LIN {X 0,Y 357.391,Z 435.676,A -85,B 0,C 180,E1 11294.259,E2 11294.259} C_VEL
LIN {X 0,Y 359.556,Z 438.789,A -85,B 0,C 180,E1 11291.438,E2 11291.438} C_VEL
LIN {X 0,Y 362.294,Z 441.241,A -85,B 0,C 180,E1 11287.88,E2 11287.88} C_VEL
LIN {X 0,Y 364.705,Z 442.533,A -85,B 0,C 180,E1 11284.575,E2 11284.575} C_VEL
LIN {X 0,Y 365.647,Z 443.721,A -85,B 0,C 180,E1 11283.201,E2 11283.201} C_VEL
LIN {X 0,Y 367.504,Z 446.415,A -85,B 0,C 180,E1 11280.039,E2 11280.039} C_VEL
LIN {X 0,Y 369.353,Z 448.083,A -85,B 0,C 180,E1 11276.876,E2 11276.876} C_VEL
LIN {X 0,Y 371.438,Z 449.318,A -85,B 0,C 180,E1 11272.974,E2 11272.974} C_VEL
LIN {X 0,Y 372.957,Z 450.083,A -85,B 0,C 180,E1 11269.742,E2 11269.742} C_VEL
LIN {X 0,Y 374.216,Z 452.056,A -85,B 0,C 180,E1 11266.292,E2 11266.292} C_VEL
LIN {X 0,Y 375.116,Z 453.423,A -85,B 0,C 180,E1 11263.095,E2 11263.095} C_VEL
LIN {X 0,Y 375.998,Z 454.396,A -85,B 0,C 180,E1 11259.644,E2 11259.644} C_VEL
LIN {X 0,Y 376.539,Z 454.956,A -85,B 0,C 180,E1 11256.097,E2 11256.097} C_VEL
LIN {X 0,Y 376.912,Z 455.194,A -85,B 0,C 180,E1 11252.737,E2 11252.737} C_VEL
LIN {X 0,Y 376.943,Z 455.24,A -85,B 0,C 180,E1 11249.088,E2 11249.088} C_VEL
LIN {X 0,Y 376.782,Z 455.124,A -85,B 0,C 180,E1 11245.739,E2 11245.739} C_VEL
LIN {X 0,Y 376.258,Z 454.711,A -85,B 0,C 180,E1 11242.057,E2 11242.057} C_VEL
LIN {X 0,Y 375.613,Z 454.001,A -85,B 0,C 180,E1 11238.795,E2 11238.795} C_VEL
LIN {X 0,Y 374.6,Z 452.721,A -85,B 0,C 180,E1 11235.066,E2 11235.066} C_VEL
LIN {X 0,Y 373.634,Z 450.999,A -85,B 0,C 180,E1 11232.077,E2 11232.077} C_VEL
LIN {X 0,Y 372.596,Z 449.782,A -85,B 0,C 180,E1 11229.419,E2 11229.419} C_VEL
LIN {X 0,Y 370.725,Z 448.948,A -85,B 0,C 180,E1 11225.63,E2 11225.63} C_VEL
LIN {X 0,Y 368.919,Z 447.787,A -85,B 0,C 180,E1 11222.391,E2 11222.391} C_VEL
LIN {X 0,Y 366.884,Z 445.572,A -85,B 0,C 180,E1 11218.816,E2 11218.816} C_VEL
LIN {X 0,Y 364.823,Z 442.577,A -85,B 0,C 180,E1 11215.582,E2 11215.582} C_VEL
LIN {X 0,Y 362.364,Z 441.294,A -85,B 0,C 180,E1 11212.227,E2 11212.227} C_VEL
LIN {X 0,Y 359.63,Z 438.864,A -85,B 0,C 180,E1 11208.648,E2 11208.648} C_VEL
LIN {X 0,Y 357.486,Z 435.84,A -85,B 0,C 180,E1 11205.86,E2 11205.86} C_VEL
LIN {X 0,Y 355.327,Z 434.438,A -85,B 0,C 180,E1 11203.361,E2 11203.361} C_VEL
LIN {X 0,Y 352.433,Z 432.047,A -85,B 0,C 180,E1 11200.091,E2 11200.091} C_VEL
LIN {X 0,Y 350.007,Z 428.702,A -85,B 0,C 180,E1 11197.273,E2 11197.273} C_VEL
LIN {X 0,Y 348.432,Z 427.598,A -85,B 0,C 180,E1 11195.628,E2 11195.628} C_VEL
LIN {X 0,Y 345.313,Z 425.117,A -85,B 0,C 180,E1 11192.389,E2 11192.389} C_VEL
LIN {X 0,Y 342.845,Z 421.896,A -85,B 0,C 180,E1 11189.721,E2 11189.721} C_VEL
LIN {X 0,Y 341.776,Z 420.845,A -85,B 0,C 180,E1 11188.671,E2 11188.671} C_VEL
LIN {X 0,Y 338.023,Z 418.479,A -85,B 0,C 180,E1 11185.586,E2 11185.586} C_VEL
LIN {X 0,Y 334.266,Z 415.023,A -85,B 0,C 180,E1 11182.883,E2 11182.883} C_VEL
LIN {X 0,Y 332.281,Z 413.005,A -85,B 0,C 180,E1 11181.537,E2 11181.537} C_VEL
LIN {X 0,Y 327.822,Z 409.906,A -85,B 0,C 180,E1 11178.863,E2 11178.863} C_VEL
LIN {X 0,Y 322.978,Z 404.536,A -85,B 0,C 180,E1 11175.687,E2 11175.687} C_VEL
LIN {X 0,Y 319.536,Z 400.127,A -85,B 0,C 180,E1 11172.836,E2 11172.836} C_VEL
LIN {X 0,Y 318.657,Z 398.667,A -85,B 0,C 180,E1 11171.952,E2 11171.952} C_VEL
LIN {X 0,Y 315.762,Z 394.618,A -85,B 0,C 180,E1 11168.467,E2 11168.467} C_VEL
LIN {X 0,Y 315.284,Z 393.503,A -85,B 0,C 180,E1 11167.654,E2 11167.654} C_VEL
LIN {X 0,Y 312.928,Z 391.284,A -85,B 0,C 180,E1 11160.915,E2 11160.915} C_VEL
LIN {X 0,Y 313.352,Z 391.949,A -85,B 0,C 180,E1 11156.891,E2 11156.891} C_VEL
LIN {X 0,Y 315.434,Z 393.763,A -85,B 0,C 180,E1 11152.533,E2 11152.533} C_VEL
LIN {X 0,Y 317.844,Z 397.884,A -85,B 0,C 180,E1 11149.304,E2 11149.304} C_VEL
LIN {X 0,Y 319.163,Z 399.431,A -85,B 0,C 180,E1 11147.976,E2 11147.976} C_VEL
LIN {X 0,Y 323.04,Z 405.209,A -85,B 0,C 180,E1 11144.655,E2 11144.655} C_VEL
LIN {X 0,Y 326.338,Z 410.188,A -85,B 0,C 180,E1 11142.343,E2 11142.343} C_VEL
LIN {X 0,Y 331.124,Z 417.365,A -85,B 0,C 180,E1 11139.496,E2 11139.496} C_VEL
LIN {X 0,Y 334.176,Z 422.791,A -85,B 0,C 180,E1 11137.852,E2 11137.852} C_VEL
LIN {X 0,Y 338.881,Z 432.418,A -85,B 0,C 180,E1 11135.51,E2 11135.51} C_VEL
LIN {X 0,Y 340.966,Z 437.107,A -85,B 0,C 180,E1 11134.535,E2 11134.535} C_VEL
LIN {X 0,Y 339.393,Z 457.12,A -85,B 0,C 180,E1 11134.133,E2 11134.133} C_VEL
LIN {X 0,Y 338.344,Z 464.817,A -85,B 0,C 180,E1 11134.132,E2 11134.132} C_VEL
LIN {X 0,Y 333.991,Z 485.367,A -85,B 0,C 180,E1 11134.678,E2 11134.678} C_VEL
LIN {X 0,Y 333.138,Z 491.97,A -85,B 0,C 180,E1 11134.661,E2 11134.661} C_VEL
LIN {X 0,Y 324.438,Z 599.073,A -85,B 0,C 180,E1 11132.465,E2 11132.465} C_VEL
LIN {X 0,Y 320.784,Z 623.389,A -85,B 0,C 180,E1 11131.786,E2 11131.786} C_VEL
LIN {X 0,Y 316.917,Z 641.647,A -85,B 0,C 180,E1 11131.101,E2 11131.101} C_VEL
LIN {X 0,Y 312.027,Z 660.593,A -85,B 0,C 180,E1 11130.177,E2 11130.177} C_VEL
LIN {X 0,Y 305.137,Z 682.435,A -85,B 0,C 180,E1 11128.783,E2 11128.783} C_VEL
LIN {X 0,Y 298.819,Z 699.564,A -85,B 0,C 180,E1 11127.404,E2 11127.404} C_VEL
LIN {X 0,Y 291.032,Z 718.423,A -85,B 0,C 180,E1 11125.539,E2 11125.539} C_VEL
LIN {X 0,Y 282.813,Z 735.832,A -85,B 0,C 180,E1 11123.371,E2 11123.371} C_VEL
LIN {X 0,Y 275.348,Z 750.463,A -85,B 0,C 180,E1 11121.158,E2 11121.158} C_VEL
LIN {X 0,Y 266.704,Z 766.363,A -85,B 0,C 180,E1 11118.247,E2 11118.247} C_VEL
LIN {X 0,Y 257.927,Z 781.243,A -85,B 0,C 180,E1 11114.814,E2 11114.814} C_VEL
LIN {X 0,Y 251.129,Z 792.469,A -85,B 0,C 180,E1 11111.673,E2 11111.673} C_VEL
LIN {X 0,Y 243.527,Z 804.944,A -85,B 0,C 180,E1 11107.419,E2 11107.419} C_VEL
LIN {X 0,Y 237.187,Z 815.301,A -85,B 0,C 180,E1 11102.942,E2 11102.942} C_VEL
LIN {X 0,Y 232.588,Z 823.275,A -85,B 0,C 180,E1 11098.722,E2 11098.722} C_VEL
LIN {X 0,Y 228.301,Z 831.546,A -85,B 0,C 180,E1 11093.213,E2 11093.213} C_VEL
LIN {X 0,Y 225.883,Z 837.101,A -85,B 0,C 180,E1 11088.317,E2 11088.317} C_VEL
LIN {X 0,Y 224.59,Z 841.14,A -85,B 0,C 180,E1 11083.647,E2 11083.647} C_VEL
LIN {X 0,Y 224.047,Z 844.149,A -85,B 0,C 180,E1 11078.727,E2 11078.727} C_VEL
LIN {X 0,Y 223.976,Z 845.889,A -85,B 0,C 180,E1 11073.583,E2 11073.583} C_VEL
LIN {X 0,Y 223.996,Z 846.17,A -85,B 0,C 180,E1 11068.977,E2 11068.977} C_VEL
LIN {X 0,Y 223.975,Z 845.377,A -85,B 0,C 180,E1 11064.563,E2 11064.563} C_VEL
LIN {X 0,Y 224.105,Z 843.591,A -85,B 0,C 180,E1 11060.239,E2 11060.239} C_VEL
LIN {X 0,Y 224.692,Z 840.748,A -85,B 0,C 180,E1 11055.834,E2 11055.834} C_VEL
LIN {X 0,Y 226.189,Z 836.341,A -85,B 0,C 180,E1 11050.907,E2 11050.907} C_VEL
LIN {X 0,Y 229.32,Z 829.45,A -85,B 0,C 180,E1 11045.256,E2 11045.256} C_VEL
LIN {X 0,Y 233.115,Z 822.315,A -85,B 0,C 180,E1 11040.729,E2 11040.729} C_VEL
LIN {X 0,Y 238.319,Z 813.453,A -85,B 0,C 180,E1 11036.171,E2 11036.171} C_VEL
LIN {X 0,Y 245.397,Z 801.813,A -85,B 0,C 180,E1 11031.437,E2 11031.437} C_VEL
LIN {X 0,Y 252.004,Z 791.031,A -85,B 0,C 180,E1 11027.894,E2 11027.894} C_VEL
LIN {X 0,Y 259.516,Z 778.645,A -85,B 0,C 180,E1 11024.524,E2 11024.524} C_VEL
LIN {X 0,Y 268.58,Z 762.891,A -85,B 0,C 180,E1 11021.076,E2 11021.076} C_VEL
LIN {X 0,Y 276.219,Z 748.803,A -85,B 0,C 180,E1 11018.569,E2 11018.569} C_VEL
LIN {X 0,Y 284.677,Z 732.136,A -85,B 0,C 180,E1 11016.119,E2 11016.119} C_VEL
LIN {X 0,Y 292.974,Z 713.8,A -85,B 0,C 180,E1 11013.975,E2 11013.975} C_VEL
LIN {X 0,Y 299.637,Z 697.472,A -85,B 0,C 180,E1 11012.413,E2 11012.413} C_VEL
LIN {X 0,Y 306.898,Z 677.436,A -85,B 0,C 180,E1 11010.857,E2 11010.857} C_VEL
LIN {X 0,Y 312.927,Z 657.297,A -85,B 0,C 180,E1 11009.65,E2 11009.65} C_VEL
LIN {X 0,Y 317.385,Z 639.669,A -85,B 0,C 180,E1 11008.816,E2 11008.816} C_VEL
LIN {X 0,Y 321.862,Z 617.639,A -85,B 0,C 180,E1 11008.03,E2 11008.03} C_VEL
LIN {X 0,Y 324.697,Z 596.376,A -85,B 0,C 180,E1 11007.475,E2 11007.475} C_VEL
LIN {X 0,Y 337.198,Z 440.954,A -85,B 0,C 180,E1 11004.294,E2 11004.294} C_VEL
LIN {X 0,Y 332.27,Z 430.413,A -85,B 0,C 180,E1 11001.77,E2 11001.77} C_VEL
LIN {X 0,Y 329.221,Z 424.769,A -85,B 0,C 180,E1 11000.071,E2 11000.071} C_VEL
LIN {X 0,Y 324.819,Z 417.96,A -85,B 0,C 180,E1 10997.373,E2 10997.373} C_VEL
LIN {X 0,Y 322.038,Z 413.675,A -85,B 0,C 180,E1 10995.394,E2 10995.394} C_VEL
LIN {X 0,Y 320.191,Z 410.862,A -85,B 0,C 180,E1 10993.913,E2 10993.913} C_VEL
LIN {X 0,Y 317.215,Z 406.295,A -85,B 0,C 180,E1 10991.085,E2 10991.085} C_VEL
LIN {X 0,Y 314.43,Z 402.015,A -85,B 0,C 180,E1 10987.491,E2 10987.491} C_VEL
LIN {X 0,Y 313.894,Z 401.23,A -85,B 0,C 180,E1 10986.585,E2 10986.585} C_VEL
LIN {X 0,Y 311.948,Z 399.214,A -85,B 0,C 180,E1 10980.367,E2 10980.367} C_VEL
LIN {X 0,Y 312.409,Z 399.942,A -85,B 0,C 180,E1 10976.33,E2 10976.33} C_VEL
LIN {X 0,Y 314.345,Z 401.757,A -85,B 0,C 180,E1 10972.231,E2 10972.231} C_VEL
LIN {X 0,Y 316.81,Z 405.872,A -85,B 0,C 180,E1 10968.9,E2 10968.9} C_VEL
LIN {X 0,Y 317.925,Z 407.334,A -85,B 0,C 180,E1 10967.744,E2 10967.744} C_VEL
LIN {X 0,Y 321.341,Z 412.052,A -85,B 0,C 180,E1 10964.756,E2 10964.756} C_VEL
LIN {X 0,Y 323.001,Z 413.964,A -85,B 0,C 180,E1 10963.546,E2 10963.546} C_VEL
LIN {X 0,Y 327.432,Z 418.519,A -85,B 0,C 180,E1 10960.744,E2 10960.744} C_VEL
LIN {X 0,Y 332.012,Z 421.761,A -85,B 0,C 180,E1 10957.98,E2 10957.98} C_VEL
LIN {X 0,Y 335.685,Z 425.45,A -85,B 0,C 180,E1 10955.355,E2 10955.355} C_VEL
LIN {X 0,Y 339.012,Z 427.854,A -85,B 0,C 180,E1 10952.797,E2 10952.797} C_VEL
LIN {X 0,Y 341.404,Z 429.368,A -85,B 0,C 180,E1 10950.72,E2 10950.72} C_VEL
LIN {X 0,Y 343.92,Z 432.708,A -85,B 0,C 180,E1 10948.054,E2 10948.054} C_VEL
LIN {X 0,Y 347.005,Z 435.312,A -85,B 0,C 180,E1 10944.811,E2 10944.811} C_VEL
LIN {X 0,Y 348.8,Z 436.444,A -85,B 0,C 180,E1 10942.988,E2 10942.988} C_VEL
LIN {X 0,Y 351.378,Z 439.984,A -85,B 0,C 180,E1 10939.978,E2 10939.978} C_VEL
LIN {X 0,Y 354.275,Z 442.359,A -85,B 0,C 180,E1 10936.701,E2 10936.701} C_VEL
LIN {X 0,Y 356.338,Z 443.696,A -85,B 0,C 180,E1 10934.315,E2 10934.315} C_VEL
LIN {X 0,Y 358.427,Z 446.646,A -85,B 0,C 180,E1 10931.598,E2 10931.598} C_VEL
LIN {X 0,Y 361.149,Z 449.073,A -85,B 0,C 180,E1 10928.124,E2 10928.124} C_VEL
LIN {X 0,Y 363.636,Z 450.443,A -85,B 0,C 180,E1 10924.691,E2 10924.691} C_VEL
LIN {X 0,Y 364.634,Z 451.698,A -85,B 0,C 180,E1 10923.245,E2 10923.245} C_VEL
LIN {X 0,Y 366.572,Z 454.443,A -85,B 0,C 180,E1 10919.943,E2 10919.943} C_VEL
LIN {X 0,Y 368.437,Z 456.074,A -85,B 0,C 180,E1 10916.769,E2 10916.769} C_VEL
LIN {X 0,Y 370.437,Z 457.251,A -85,B 0,C 180,E1 10913.015,E2 10913.015} C_VEL
LIN {X 0,Y 371.948,Z 458.011,A -85,B 0,C 180,E1 10909.798,E2 10909.798} C_VEL
LIN {X 0,Y 373.203,Z 459.944,A -85,B 0,C 180,E1 10906.439,E2 10906.439} C_VEL
LIN {X 0,Y 374.126,Z 461.361,A -85,B 0,C 180,E1 10903.13,E2 10903.13} C_VEL
LIN {X 0,Y 374.962,Z 462.31,A -85,B 0,C 180,E1 10899.826,E2 10899.826} C_VEL
LIN {X 0,Y 375.545,Z 462.87,A -85,B 0,C 180,E1 10896.267,E2 10896.267} C_VEL
LIN {X 0,Y 375.886,Z 463.11,A -85,B 0,C 180,E1 10893.049,E2 10893.049} C_VEL
LIN {X 0,Y 375.975,Z 463.189,A -85,B 0,C 180,E1 10889.238,E2 10889.238} C_VEL
LIN {X 0,Y 375.805,Z 463.095,A -85,B 0,C 180,E1 10886.034,E2 10886.034} C_VEL
LIN {X 0,Y 375.311,Z 462.674,A -85,B 0,C 180,E1 10882.191,E2 10882.191} C_VEL
LIN {X 0,Y 374.684,Z 462.013,A -85,B 0,C 180,E1 10879.079,E2 10879.079} C_VEL
LIN {X 0,Y 373.799,Z 460.907,A -85,B 0,C 180,E1 10875.534,E2 10875.534} C_VEL
LIN {X 0,Y 372.703,Z 459.108,A -85,B 0,C 180,E1 10872.244,E2 10872.244} C_VEL
LIN {X 0,Y 371.727,Z 457.816,A -85,B 0,C 180,E1 10869.698,E2 10869.698} C_VEL
LIN {X 0,Y 370.035,Z 457.027,A -85,B 0,C 180,E1 10866.09,E2 10866.09} C_VEL
LIN {X 0,Y 368.084,Z 455.848,A -85,B 0,C 180,E1 10862.655,E2 10862.655} C_VEL
LIN {X 0,Y 366.169,Z 453.933,A -85,B 0,C 180,E1 10859.296,E2 10859.296} C_VEL
LIN {X 0,Y 363.981,Z 450.622,A -85,B 0,C 180,E1 10855.776,E2 10855.776} C_VEL
LIN {X 0,Y 361.582,Z 449.398,A -85,B 0,C 180,E1 10852.525,E2 10852.525} C_VEL
LIN {X 0,Y 358.842,Z 447.06,A -85,B 0,C 180,E1 10848.886,E2 10848.886} C_VEL
LIN {X 0,Y 356.443,Z 443.873,A -85,B 0,C 180,E1 10845.817,E2 10845.817} C_VEL
LIN {X 0,Y 355.498,Z 442.991,A -85,B 0,C 180,E1 10844.638,E2 10844.638} C_VEL
LIN {X 0,Y 352.409,Z 440.929,A -85,B 0,C 180,E1 10841.165,E2 10841.165} C_VEL
LIN {X 0,Y 349.883,Z 438.191,A -85,B 0,C 180,E1 10838.325,E2 10838.325} C_VEL
LIN {X 0,Y 348.298,Z 435.966,A -85,B 0,C 180,E1 10836.458,E2 10836.458} C_VEL
LIN {X 0,Y 345.092,Z 433.842,A -85,B 0,C 180,E1 10833.203,E2 10833.203} C_VEL
LIN {X 0,Y 342.244,Z 430.64,A -85,B 0,C 180,E1 10830.148,E2 10830.148} C_VEL
LIN {X 0,Y 340.87,Z 428.854,A -85,B 0,C 180,E1 10828.754,E2 10828.754} C_VEL
LIN {X 0,Y 336.984,Z 426.486,A -85,B 0,C 180,E1 10825.582,E2 10825.582} C_VEL
LIN {X 0,Y 333.203,Z 423.143,A -85,B 0,C 180,E1 10822.876,E2 10822.876} C_VEL
LIN {X 0,Y 330.785,Z 420.741,A -85,B 0,C 180,E1 10821.267,E2 10821.267} C_VEL
LIN {X 0,Y 326.293,Z 417.595,A -85,B 0,C 180,E1 10818.583,E2 10818.583} C_VEL
LIN {X 0,Y 321.458,Z 412.16,A -85,B 0,C 180,E1 10815.33,E2 10815.33} C_VEL
LIN {X 0,Y 318.01,Z 407.503,A -85,B 0,C 180,E1 10812.345,E2 10812.345} C_VEL
LIN {X 0,Y 317.151,Z 406.22,A -85,B 0,C 180,E1 10811.456,E2 10811.456} C_VEL
LIN {X 0,Y 314.495,Z 402.173,A -85,B 0,C 180,E1 10808.041,E2 10808.041} C_VEL
LIN {X 0,Y 314.078,Z 401.333,A -85,B 0,C 180,E1 10807.316,E2 10807.316} C_VEL
LIN {X 0,Y 311.953,Z 399.225,A -85,B 0,C 180,E1 10800.918,E2 10800.918} C_VEL
LIN {X 0,Y 312.376,Z 399.905,A -85,B 0,C 180,E1 10796.881,E2 10796.881} C_VEL
LIN {X 0,Y 314.331,Z 401.739,A -85,B 0,C 180,E1 10792.69,E2 10792.69} C_VEL
LIN {X 0,Y 316.871,Z 405.954,A -85,B 0,C 180,E1 10789.271,E2 10789.271} C_VEL
LIN {X 0,Y 317.9,Z 407.32,A -85,B 0,C 180,E1 10788.203,E2 10788.203} C_VEL
LIN {X 0,Y 321.483,Z 412.758,A -85,B 0,C 180,E1 10785.04,E2 10785.04} C_VEL
LIN {X 0,Y 324.755,Z 417.859,A -85,B 0,C 180,E1 10782.67,E2 10782.67} C_VEL
LIN {X 0,Y 329.149,Z 424.639,A -85,B 0,C 180,E1 10779.971,E2 10779.971} C_VEL
LIN {X 0,Y 332.193,Z 430.266,A -85,B 0,C 180,E1 10778.271,E2 10778.271} C_VEL
LIN {X 0,Y 337.032,Z 440.583,A -85,B 0,C 180,E1 10775.786,E2 10775.786} C_VEL
LIN {X 0,Y 337.216,Z 441.414,A -85,B 0,C 180,E1 10775.676,E2 10775.676} C_VEL
LIN {X 0,Y 333.138,Z 491.97,A -85,B 0,C 180,E1 10774.661,E2 10774.661} C_VEL
LIN {X 0,Y 332.088,Z 499.666,A -85,B 0,C 180,E1 10774.662,E2 10774.662} C_VEL
LIN {X 0,Y 327.745,Z 520.207,A -85,B 0,C 180,E1 10775.234,E2 10775.234} C_VEL
LIN {X 0,Y 326.89,Z 526.81,A -85,B 0,C 180,E1 10775.219,E2 10775.219} C_VEL
LIN {X 0,Y 320.737,Z 599.443,A -85,B 0,C 180,E1 10773.723,E2 10773.723} C_VEL
LIN {X 0,Y 317.015,Z 623.378,A -85,B 0,C 180,E1 10773.058,E2 10773.058} C_VEL
LIN {X 0,Y 312.936,Z 642.102,A -85,B 0,C 180,E1 10772.362,E2 10772.362} C_VEL
LIN {X 0,Y 307.544,Z 662.32,A -85,B 0,C 180,E1 10771.375,E2 10771.375} C_VEL
LIN {X 0,Y 301.018,Z 682.183,A -85,B 0,C 180,E1 10770.102,E2 10770.102} C_VEL
LIN {X 0,Y 294.664,Z 698.957,A -85,B 0,C 180,E1 10768.767,E2 10768.767} C_VEL
LIN {X 0,Y 287.158,Z 716.63,A -85,B 0,C 180,E1 10767.047,E2 10767.047} C_VEL
LIN {X 0,Y 278.254,Z 735.093,A -85,B 0,C 180,E1 10764.793,E2 10764.793} C_VEL
LIN {X 0,Y 270.569,Z 749.654,A -85,B 0,C 180,E1 10762.607,E2 10762.607} C_VEL
LIN {X 0,Y 261.937,Z 764.943,A -85,B 0,C 180,E1 10759.827,E2 10759.827} C_VEL
LIN {X 0,Y 252.731,Z 780.039,A -85,B 0,C 180,E1 10756.383,E2 10756.383} C_VEL
LIN {X 0,Y 245.462,Z 791.493,A -85,B 0,C 180,E1 10753.181,E2 10753.181} C_VEL
LIN {X 0,Y 237.773,Z 803.479,A -85,B 0,C 180,E1 10749.105,E2 10749.105} C_VEL
LIN {X 0,Y 230.588,Z 814.544,A -85,B 0,C 180,E1 10744.311,E2 10744.311} C_VEL
LIN {X 0,Y 225.666,Z 822.493,A -85,B 0,C 180,E1 10740.043,E2 10740.043} C_VEL
LIN {X 0,Y 221.098,Z 830.662,A -85,B 0,C 180,E1 10734.584,E2 10734.584} C_VEL
LIN {X 0,Y 218.107,Z 836.846,A -85,B 0,C 180,E1 10728.994,E2 10728.994} C_VEL
LIN {X 0,Y 216.678,Z 840.887,A -85,B 0,C 180,E1 10724.156,E2 10724.156} C_VEL
LIN {X 0,Y 216.059,Z 843.898,A -85,B 0,C 180,E1 10719.052,E2 10719.052} C_VEL
LIN {X 0,Y 215.978,Z 845.64,A -85,B 0,C 180,E1 10713.716,E2 10713.716} C_VEL
LIN {X 0,Y 215.999,Z 845.922,A -85,B 0,C 180,E1 10708.939,E2 10708.939} C_VEL
LIN {X 0,Y 215.977,Z 845.146,A -85,B 0,C 180,E1 10704.421,E2 10704.421} C_VEL
LIN {X 0,Y 216.133,Z 843.339,A -85,B 0,C 180,E1 10699.875,E2 10699.875} C_VEL
LIN {X 0,Y 216.791,Z 840.495,A -85,B 0,C 180,E1 10695.306,E2 10695.306} C_VEL
LIN {X 0,Y 218.444,Z 836.086,A -85,B 0,C 180,E1 10690.202,E2 10690.202} C_VEL
LIN {X 0,Y 221.871,Z 829.144,A -85,B 0,C 180,E1 10684.329,E2 10684.329} C_VEL
LIN {X 0,Y 226.01,Z 821.916,A -85,B 0,C 180,E1 10679.618,E2 10679.618} C_VEL
LIN {X 0,Y 231.575,Z 813.045,A -85,B 0,C 180,E1 10674.954,E2 10674.954} C_VEL
LIN {X 0,Y 238.967,Z 801.555,A -85,B 0,C 180,E1 10670.197,E2 10670.197} C_VEL
LIN {X 0,Y 245.924,Z 790.774,A -85,B 0,C 180,E1 10666.6,E2 10666.6} C_VEL
LIN {X 0,Y 253.76,Z 778.433,A -85,B 0,C 180,E1 10663.205,E2 10663.205} C_VEL
LIN {X 0,Y 263.239,Z 762.635,A -85,B 0,C 180,E1 10659.724,E2 10659.724} C_VEL
LIN {X 0,Y 271.174,Z 748.548,A -85,B 0,C 180,E1 10657.212,E2 10657.212} C_VEL
LIN {X 0,Y 279.935,Z 731.882,A -85,B 0,C 180,E1 10654.767,E2 10654.767} C_VEL
LIN {X 0,Y 288.501,Z 713.547,A -85,B 0,C 180,E1 10652.633,E2 10652.633} C_VEL
LIN {X 0,Y 295.013,Z 698.088,A -85,B 0,C 180,E1 10651.158,E2 10651.158} C_VEL
LIN {X 0,Y 301.739,Z 680.21,A -85,B 0,C 180,E1 10649.755,E2 10649.755} C_VEL
LIN {X 0,Y 308.412,Z 659.201,A -85,B 0,C 180,E1 10648.461,E2 10648.461} C_VEL
LIN {X 0,Y 313.144,Z 641.241,A -85,B 0,C 180,E1 10647.603,E2 10647.603} C_VEL
LIN {X 0,Y 317.327,Z 621.825,A -85,B 0,C 180,E1 10646.891,E2 10646.891} C_VEL
LIN {X 0,Y 320.845,Z 598.276,A -85,B 0,C 180,E1 10646.251,E2 10646.251} C_VEL
LIN {X 0,Y 329.877,Z 490.536,A -85,B 0,C 180,E1 10644.053,E2 10644.053} C_VEL
LIN {X 0,Y 333.578,Z 445.2,A -85,B 0,C 180,E1 10643.12,E2 10643.12} C_VEL
LIN {X 0,Y 329.131,Z 435.484,A -85,B 0,C 180,E1 10640.68,E2 10640.68} C_VEL
LIN {X 0,Y 325.729,Z 429.591,A -85,B 0,C 180,E1 10638.663,E2 10638.663} C_VEL
LIN {X 0,Y 321.157,Z 422.258,A -85,B 0,C 180,E1 10635.53,E2 10635.53} C_VEL
LIN {X 0,Y 318.791,Z 418.549,A -85,B 0,C 180,E1 10633.605,E2 10633.605} C_VEL
LIN {X 0,Y 315.899,Z 414.011,A -85,B 0,C 180,E1 10630.763,E2 10630.763} C_VEL
LIN {X 0,Y 313.231,Z 409.703,A -85,B 0,C 180,E1 10627.151,E2 10627.151} C_VEL
LIN {X 0,Y 312.506,Z 408.918,A -85,B 0,C 180,E1 10625.876,E2 10625.876} C_VEL
LIN {X 0,Y 310.963,Z 407.159,A -85,B 0,C 180,E1 10620.184,E2 10620.184} C_VEL
LIN {X 0,Y 311.544,Z 408.033,A -85,B 0,C 180,E1 10615.951,E2 10615.951} C_VEL
LIN {X 0,Y 313.198,Z 409.588,A -85,B 0,C 180,E1 10612.479,E2 10612.479} C_VEL
LIN {X 0,Y 315.671,Z 413.761,A -85,B 0,C 180,E1 10609.045,E2 10609.045} C_VEL
LIN {X 0,Y 316.669,Z 415.215,A -85,B 0,C 180,E1 10607.972,E2 10607.972} C_VEL
LIN {X 0,Y 320.03,Z 419.855,A -85,B 0,C 180,E1 10604.971,E2 10604.971} C_VEL
LIN {X 0,Y 321.895,Z 422.169,A -85,B 0,C 180,E1 10603.581,E2 10603.581} C_VEL
LIN {X 0,Y 326.487,Z 426.645,A -85,B 0,C 180,E1 10600.686,E2 10600.686} C_VEL
LIN {X 0,Y 330.647,Z 429.602,A -85,B 0,C 180,E1 10598.175,E2 10598.175} C_VEL
LIN {X 0,Y 334.524,Z 433.377,A -85,B 0,C 180,E1 10595.452,E2 10595.452} C_VEL
LIN {X 0,Y 337.872,Z 435.755,A -85,B 0,C 180,E1 10592.888,E2 10592.888} C_VEL
LIN {X 0,Y 340.221,Z 437.245,A -85,B 0,C 180,E1 10590.897,E2 10590.897} C_VEL
LIN {X 0,Y 342.843,Z 440.641,A -85,B 0,C 180,E1 10588.139,E2 10588.139} C_VEL
LIN {X 0,Y 345.949,Z 443.234,A -85,B 0,C 180,E1 10584.875,E2 10584.875} C_VEL
LIN {X 0,Y 347.674,Z 444.334,A -85,B 0,C 180,E1 10583.148,E2 10583.148} C_VEL
LIN {X 0,Y 350.325,Z 447.923,A -85,B 0,C 180,E1 10580.046,E2 10580.046} C_VEL
LIN {X 0,Y 353.066,Z 450.187,A -85,B 0,C 180,E1 10576.938,E2 10576.938} C_VEL
LIN {X 0,Y 355.189,Z 451.538,A -85,B 0,C 180,E1 10574.501,E2 10574.501} C_VEL
LIN {X 0,Y 357.301,Z 454.503,A -85,B 0,C 180,E1 10571.758,E2 10571.758} C_VEL
LIN {X 0,Y 359.934,Z 456.869,A -85,B 0,C 180,E1 10568.43,E2 10568.43} C_VEL
LIN {X 0,Y 362.569,Z 458.35,A -85,B 0,C 180,E1 10564.808,E2 10564.808} C_VEL
LIN {X 0,Y 363.889,Z 460.154,A -85,B 0,C 180,E1 10562.776,E2 10562.776} C_VEL
LIN {X 0,Y 365.641,Z 462.464,A -85,B 0,C 180,E1 10559.846,E2 10559.846} C_VEL
LIN {X 0,Y 367.515,Z 464.063,A -85,B 0,C 180,E1 10556.672,E2 10556.672} C_VEL
LIN {X 0,Y 369.494,Z 465.208,A -85,B 0,C 180,E1 10552.933,E2 10552.933} C_VEL
LIN {X 0,Y 370.95,Z 465.946,A -85,B 0,C 180,E1 10549.832,E2 10549.832} C_VEL
LIN {X 0,Y 372.219,Z 467.889,A -85,B 0,C 180,E1 10546.469,E2 10546.469} C_VEL
LIN {X 0,Y 373.136,Z 469.299,A -85,B 0,C 180,E1 10543.165,E2 10543.165} C_VEL
LIN {X 0,Y 373.974,Z 470.247,A -85,B 0,C 180,E1 10539.852,E2 10539.852} C_VEL
LIN {X 0,Y 374.565,Z 470.809,A -85,B 0,C 180,E1 10536.283,E2 10536.283} C_VEL
LIN {X 0,Y 374.886,Z 471.047,A -85,B 0,C 180,E1 10533.211,E2 10533.211} C_VEL
LIN {X 0,Y 375.024,Z 471.146,A -85,B 0,C 180,E1 10529.542,E2 10529.542} C_VEL
LIN {X 0,Y 374.842,Z 471.044,A -85,B 0,C 180,E1 10526.33,E2 10526.33} C_VEL
LIN {X 0,Y 374.498,Z 470.672,A -85,B 0,C 180,E1 10522.792,E2 10522.792} C_VEL
LIN {X 0,Y 373.763,Z 470.044,A -85,B 0,C 180,E1 10519.363,E2 10519.363} C_VEL
LIN {X 0,Y 372.941,Z 468.996,A -85,B 0,C 180,E1 10515.879,E2 10515.879} C_VEL
LIN {X 0,Y 371.798,Z 467.254,A -85,B 0,C 180,E1 10512.471,E2 10512.471} C_VEL
LIN {X 0,Y 370.863,Z 465.878,A -85,B 0,C 180,E1 10509.978,E2 10509.978} C_VEL
LIN {X 0,Y 369.342,Z 465.136,A -85,B 0,C 180,E1 10506.72,E2 10506.72} C_VEL
LIN {X 0,Y 367.397,Z 463.988,A -85,B 0,C 180,E1 10503.144,E2 10503.144} C_VEL
LIN {X 0,Y 365.611,Z 462.434,A -85,B 0,C 180,E1 10500.102,E2 10500.102} C_VEL
LIN {X 0,Y 363.687,Z 459.791,A -85,B 0,C 180,E1 10496.833,E2 10496.833} C_VEL
LIN {X 0,Y 362.569,Z 458.35,A -85,B 0,C 180,E1 10495.192,E2 10495.192} C_VEL
LIN {X 0,Y 359.889,Z 456.839,A -85,B 0,C 180,E1 10491.515,E2 10491.515} C_VEL
LIN {X 0,Y 357.301,Z 454.503,A -85,B 0,C 180,E1 10488.242,E2 10488.242} C_VEL
LIN {X 0,Y 355.189,Z 451.538,A -85,B 0,C 180,E1 10485.499,E2 10485.499} C_VEL
LIN {X 0,Y 352.071,Z 449.434,A -85,B 0,C 180,E1 10481.865,E2 10481.865} C_VEL
LIN {X 0,Y 348.984,Z 446.395,A -85,B 0,C 180,E1 10478.442,E2 10478.442} C_VEL
LIN {X 0,Y 347.23,Z 443.882,A -85,B 0,C 180,E1 10476.383,E2 10476.383} C_VEL
LIN {X 0,Y 344.009,Z 441.766,A -85,B 0,C 180,E1 10473.122,E2 10473.122} C_VEL
LIN {X 0,Y 341.073,Z 438.521,A -85,B 0,C 180,E1 10469.988,E2 10469.988} C_VEL
LIN {X 0,Y 339.548,Z 436.654,A -85,B 0,C 180,E1 10468.492,E2 10468.492} C_VEL
LIN {X 0,Y 335.686,Z 434.306,A -85,B 0,C 180,E1 10465.398,E2 10465.398} C_VEL
LIN {X 0,Y 331.877,Z 430.971,A -85,B 0,C 180,E1 10462.683,E2 10462.683} C_VEL
LIN {X 0,Y 329.296,Z 428.475,A -85,B 0,C 180,E1 10460.995,E2 10460.995} C_VEL
LIN {X 0,Y 324.353,Z 424.912,A -85,B 0,C 180,E1 10458.047,E2 10458.047} C_VEL
LIN {X 0,Y 320.03,Z 419.855,A -85,B 0,C 180,E1 10455.029,E2 10455.029} C_VEL
LIN {X 0,Y 316.669,Z 415.215,A -85,B 0,C 180,E1 10452.028,E2 10452.028} C_VEL
LIN {X 0,Y 315.671,Z 413.761,A -85,B 0,C 180,E1 10450.955,E2 10450.955} C_VEL
LIN {X 0,Y 313.198,Z 409.588,A -85,B 0,C 180,E1 10447.521,E2 10447.521} C_VEL
LIN {X 0,Y 311.003,Z 407.221,A -85,B 0,C 180,E1 10441.29,E2 10441.29} C_VEL
LIN {X 0,Y 311.224,Z 407.605,A -85,B 0,C 180,E1 10437.606,E2 10437.606} C_VEL
LIN {X 0,Y 313.184,Z 409.568,A -85,B 0,C 180,E1 10432.94,E2 10432.94} C_VEL
LIN {X 0,Y 315.73,Z 413.841,A -85,B 0,C 180,E1 10429.416,E2 10429.416} C_VEL
LIN {X 0,Y 316.643,Z 415.2,A -85,B 0,C 180,E1 10428.433,E2 10428.433} C_VEL
LIN {X 0,Y 319.94,Z 420.308,A -85,B 0,C 180,E1 10425.429,E2 10425.429} C_VEL
LIN {X 0,Y 323.309,Z 425.726,A -85,B 0,C 180,E1 10422.915,E2 10422.915} C_VEL
LIN {X 0,Y 327.548,Z 432.552,A -85,B 0,C 180,E1 10420.241,E2 10420.241} C_VEL
LIN {X 0,Y 330.447,Z 438.243,A -85,B 0,C 180,E1 10418.57,E2 10418.57} C_VEL
LIN {X 0,Y 333.622,Z 445.496,A -85,B 0,C 180,E1 10416.847,E2 10416.847} C_VEL
LIN {X 0,Y 326.89,Z 526.81,A -85,B 0,C 180,E1 10415.219,E2 10415.219} C_VEL
LIN {X 0,Y 325.843,Z 534.503,A -85,B 0,C 180,E1 10415.221,E2 10415.221} C_VEL
LIN {X 0,Y 321.522,Z 555.036,A -85,B 0,C 180,E1 10415.816,E2 10415.816} C_VEL
LIN {X 0,Y 320.65,Z 561.641,A -85,B 0,C 180,E1 10415.808,E2 10415.808} C_VEL
LIN {X 0,Y 316.921,Z 602.279,A -85,B 0,C 180,E1 10414.953,E2 10414.953} C_VEL
LIN {X 0,Y 313.188,Z 624.447,A -85,B 0,C 180,E1 10414.325,E2 10414.325} C_VEL
LIN {X 0,Y 309.072,Z 642.714,A -85,B 0,C 180,E1 10413.647,E2 10413.647} C_VEL
LIN {X 0,Y 303.384,Z 663.337,A -85,B 0,C 180,E1 10412.643,E2 10412.643} C_VEL
LIN {X 0,Y 296.732,Z 682.819,A -85,B 0,C 180,E1 10411.392,E2 10411.392} C_VEL
LIN {X 0,Y 290.178,Z 699.573,A -85,B 0,C 180,E1 10410.062,E2 10410.062} C_VEL
LIN {X 0,Y 281.874,Z 718.44,A -85,B 0,C 180,E1 10408.215,E2 10408.215} C_VEL
LIN {X 0,Y 273.029,Z 735.94,A -85,B 0,C 180,E1 10406.041,E2 10406.041} C_VEL
LIN {X 0,Y 265.038,Z 750.506,A -85,B 0,C 180,E1 10403.832,E2 10403.832} C_VEL
LIN {X 0,Y 255.434,Z 766.758,A -85,B 0,C 180,E1 10400.807,E2 10400.807} C_VEL
LIN {X 0,Y 246.572,Z 780.585,A -85,B 0,C 180,E1 10397.561,E2 10397.561} C_VEL
LIN {X 0,Y 239.011,Z 791.954,A -85,B 0,C 180,E1 10394.314,E2 10394.314} C_VEL
LIN {X 0,Y 230.568,Z 804.428,A -85,B 0,C 180,E1 10389.925,E2 10389.925} C_VEL
LIN {X 0,Y 223.444,Z 814.786,A -85,B 0,C 180,E1 10385.256,E2 10385.256} C_VEL
LIN {X 0,Y 218.26,Z 822.67,A -85,B 0,C 180,E1 10380.868,E2 10380.868} C_VEL
LIN {X 0,Y 213.425,Z 830.721,A -85,B 0,C 180,E1 10375.233,E2 10375.233} C_VEL
LIN {X 0,Y 210.36,Z 836.591,A -85,B 0,C 180,E1 10369.722,E2 10369.722} C_VEL
LIN {X 0,Y 208.779,Z 840.634,A -85,B 0,C 180,E1 10364.703,E2 10364.703} C_VEL
LIN {X 0,Y 208.078,Z 843.646,A -85,B 0,C 180,E1 10359.403,E2 10359.403} C_VEL
LIN {X 0,Y 207.98,Z 845.391,A -85,B 0,C 180,E1 10353.859,E2 10353.859} C_VEL
LIN {X 0,Y 208.002,Z 845.674,A -85,B 0,C 180,E1 10348.898,E2 10348.898} C_VEL
LIN {X 0,Y 207.98,Z 844.896,A -85,B 0,C 180,E1 10344.206,E2 10344.206} C_VEL
LIN {X 0,Y 208.163,Z 843.088,A -85,B 0,C 180,E1 10339.484,E2 10339.484} C_VEL
LIN {X 0,Y 208.905,Z 840.241,A -85,B 0,C 180,E1 10334.738,E2 10334.738} C_VEL
LIN {X 0,Y 210.73,Z 835.831,A -85,B 0,C 180,E1 10329.445,E2 10329.445} C_VEL
LIN {X 0,Y 214.422,Z 828.936,A -85,B 0,C 180,E1 10323.408,E2 10323.408} C_VEL
LIN {X 0,Y 218.809,Z 821.801,A -85,B 0,C 180,E1 10318.606,E2 10318.606} C_VEL
LIN {X 0,Y 224.481,Z 813.287,A -85,B 0,C 180,E1 10313.99,E2 10313.99} C_VEL
LIN {X 0,Y 232.657,Z 801.298,A -85,B 0,C 180,E1 10308.89,E2 10308.89} C_VEL
LIN {X 0,Y 239.978,Z 790.517,A -85,B 0,C 180,E1 10305.242,E2 10305.242} C_VEL
LIN {X 0,Y 248.174,Z 778.176,A -85,B 0,C 180,E1 10301.814,E2 10301.814} C_VEL
LIN {X 0,Y 258.099,Z 762.305,A -85,B 0,C 180,E1 10298.304,E2 10298.304} C_VEL
LIN {X 0,Y 266.29,Z 748.293,A -85,B 0,C 180,E1 10295.805,E2 10295.805} C_VEL
LIN {X 0,Y 275.356,Z 731.628,A -85,B 0,C 180,E1 10293.37,E2 10293.37} C_VEL
LIN {X 0,Y 284.191,Z 713.294,A -85,B 0,C 180,E1 10291.25,E2 10291.25} C_VEL
LIN {X 0,Y 291.037,Z 697.497,A -85,B 0,C 180,E1 10289.76,E2 10289.76} C_VEL
LIN {X 0,Y 298.549,Z 677.986,A -85,B 0,C 180,E1 10288.264,E2 10288.264} C_VEL
LIN {X 0,Y 305.08,Z 657.455,A -85,B 0,C 180,E1 10287.051,E2 10287.051} C_VEL
LIN {X 0,Y 309.846,Z 639.584,A -85,B 0,C 180,E1 10286.225,E2 10286.225} C_VEL
LIN {X 0,Y 314.536,Z 617.752,A -85,B 0,C 180,E1 10285.463,E2 10285.463} C_VEL
LIN {X 0,Y 317.592,Z 595.981,A -85,B 0,C 180,E1 10284.904,E2 10284.904} C_VEL
LIN {X 0,Y 330.118,Z 449.521,A -85,B 0,C 180,E1 10281.932,E2 10281.932} C_VEL
LIN {X 0,Y 326.167,Z 440.815,A -85,B 0,C 180,E1 10279.613,E2 10279.613} C_VEL
LIN {X 0,Y 321.808,Z 433.477,A -85,B 0,C 180,E1 10276.795,E2 10276.795} C_VEL
LIN {X 0,Y 318.724,Z 428.405,A -85,B 0,C 180,E1 10274.442,E2 10274.442} C_VEL
LIN {X 0,Y 317.001,Z 425.719,A -85,B 0,C 180,E1 10272.941,E2 10272.941} C_VEL
LIN {X 0,Y 314.592,Z 421.725,A -85,B 0,C 180,E1 10270.437,E2 10270.437} C_VEL
LIN {X 0,Y 312.043,Z 417.391,A -85,B 0,C 180,E1 10266.809,E2 10266.809} C_VEL
LIN {X 0,Y 310.007,Z 415.114,A -85,B 0,C 180,E1 10260.554,E2 10260.554} C_VEL
LIN {X 0,Y 310.36,Z 415.727,A -85,B 0,C 180,E1 10256.676,E2 10256.676} C_VEL
LIN {X 0,Y 312.057,Z 417.417,A -85,B 0,C 180,E1 10252.729,E2 10252.729} C_VEL
LIN {X 0,Y 314.577,Z 421.694,A -85,B 0,C 180,E1 10249.145,E2 10249.145} C_VEL
LIN {X 0,Y 318.837,Z 427.764,A -85,B 0,C 180,E1 10245.099,E2 10245.099} C_VEL
LIN {X 0,Y 324.25,Z 433.798,A -85,B 0,C 180,E1 10241.388,E2 10241.388} C_VEL
LIN {X 0,Y 329.162,Z 437.327,A -85,B 0,C 180,E1 10238.436,E2 10238.436} C_VEL
LIN {X 0,Y 333.142,Z 441.105,A -85,B 0,C 180,E1 10235.721,E2 10235.721} C_VEL
LIN {X 0,Y 336.51,Z 443.533,A -85,B 0,C 180,E1 10233.152,E2 10233.152} C_VEL
LIN {X 0,Y 339.026,Z 445.119,A -85,B 0,C 180,E1 10231.075,E2 10231.075} C_VEL
LIN {X 0,Y 341.766,Z 448.573,A -85,B 0,C 180,E1 10228.224,E2 10228.224} C_VEL
LIN {X 0,Y 345.041,Z 451.244,A -85,B 0,C 180,E1 10224.784,E2 10224.784} C_VEL
LIN {X 0,Y 346.6,Z 452.326,A -85,B 0,C 180,E1 10223.231,E2 10223.231} C_VEL
LIN {X 0,Y 349.286,Z 455.875,A -85,B 0,C 180,E1 10220.099,E2 10220.099} C_VEL
LIN {X 0,Y 352.143,Z 458.185,A -85,B 0,C 180,E1 10216.861,E2 10216.861} C_VEL
LIN {X 0,Y 354.081,Z 459.449,A -85,B 0,C 180,E1 10214.635,E2 10214.635} C_VEL
LIN {X 0,Y 356.178,Z 462.359,A -85,B 0,C 180,E1 10211.92,E2 10211.92} C_VEL
LIN {X 0,Y 358.709,Z 464.678,A -85,B 0,C 180,E1 10208.697,E2 10208.697} C_VEL
LIN {X 0,Y 361.431,Z 466.223,A -85,B 0,C 180,E1 10205.03,E2 10205.03} C_VEL
LIN {X 0,Y 362.367,Z 467.299,A -85,B 0,C 180,E1 10203.683,E2 10203.683} C_VEL
LIN {X 0,Y 364.491,Z 470.261,A -85,B 0,C 180,E1 10200.131,E2 10200.131} C_VEL
LIN {X 0,Y 366.248,Z 471.832,A -85,B 0,C 180,E1 10197.123,E2 10197.123} C_VEL
LIN {X 0,Y 368.265,Z 473.022,A -85,B 0,C 180,E1 10193.522,E2 10193.522} C_VEL
LIN {X 0,Y 369.787,Z 473.742,A -85,B 0,C 180,E1 10190.242,E2 10190.242} C_VEL
LIN {X 0,Y 370.739,Z 475.083,A -85,B 0,C 180,E1 10187.743,E2 10187.743} C_VEL
LIN {X 0,Y 371.829,Z 476.805,A -85,B 0,C 180,E1 10184.482,E2 10184.482} C_VEL
LIN {X 0,Y 372.723,Z 477.901,A -85,B 0,C 180,E1 10180.942,E2 10180.942} C_VEL
LIN {X 0,Y 373.368,Z 478.559,A -85,B 0,C 180,E1 10177.763,E2 10177.763} C_VEL
LIN {X 0,Y 373.849,Z 478.975,A -85,B 0,C 180,E1 10173.984,E2 10173.984} C_VEL
LIN {X 0,Y 374.021,Z 479.069,A -85,B 0,C 180,E1 10170.766,E2 10170.766} C_VEL
LIN {X 0,Y 373.928,Z 478.991,A -85,B 0,C 180,E1 10166.935,E2 10166.935} C_VEL
LIN {X 0,Y 373.6,Z 478.773,A -85,B 0,C 180,E1 10163.855,E2 10163.855} C_VEL
LIN {X 0,Y 373.039,Z 478.208,A -85,B 0,C 180,E1 10160.279,E2 10160.279} C_VEL
LIN {X 0,Y 372.187,Z 477.299,A -85,B 0,C 180,E1 10156.959,E2 10156.959} C_VEL
LIN {X 0,Y 371.248,Z 475.865,A -85,B 0,C 180,E1 10153.574,E2 10153.574} C_VEL
LIN {X 0,Y 370.01,Z 473.919,A -85,B 0,C 180,E1 10150.259,E2 10150.259} C_VEL
LIN {X 0,Y 368.562,Z 473.168,A -85,B 0,C 180,E1 10147.174,E2 10147.174} C_VEL
LIN {X 0,Y 366.611,Z 472.065,A -85,B 0,C 180,E1 10143.451,E2 10143.451} C_VEL
LIN {X 0,Y 364.713,Z 470.482,A -85,B 0,C 180,E1 10140.251,E2 10140.251} C_VEL
LIN {X 0,Y 362.95,Z 468.255,A -85,B 0,C 180,E1 10137.321,E2 10137.321} C_VEL
LIN {X 0,Y 361.503,Z 466.256,A -85,B 0,C 180,E1 10135.074,E2 10135.074} C_VEL
LIN {X 0,Y 358.71,Z 464.678,A -85,B 0,C 180,E1 10131.303,E2 10131.303} C_VEL
LIN {X 0,Y 356.178,Z 462.359,A -85,B 0,C 180,E1 10128.08,E2 10128.08} C_VEL
LIN {X 0,Y 354.046,Z 459.386,A -85,B 0,C 180,E1 10125.317,E2 10125.317} C_VEL
LIN {X 0,Y 350.851,Z 457.223,A -85,B 0,C 180,E1 10121.606,E2 10121.606} C_VEL
LIN {X 0,Y 347.857,Z 454.292,A -85,B 0,C 180,E1 10118.31,E2 10118.31} C_VEL
LIN {X 0,Y 345.961,Z 451.709,A -85,B 0,C 180,E1 10116.127,E2 10116.127} C_VEL
LIN {X 0,Y 342.927,Z 449.689,A -85,B 0,C 180,E1 10113.04,E2 10113.04} C_VEL
LIN {X 0,Y 340.052,Z 446.61,A -85,B 0,C 180,E1 10109.99,E2 10109.99} C_VEL
LIN {X 0,Y 338.43,Z 444.557,A -85,B 0,C 180,E1 10108.402,E2 10108.402} C_VEL
LIN {X 0,Y 334.517,Z 442.217,A -85,B 0,C 180,E1 10105.304,E2 10105.304} C_VEL
LIN {X 0,Y 330.685,Z 438.933,A -85,B 0,C 180,E1 10102.581,E2 10102.581} C_VEL
LIN {X 0,Y 327.816,Z 436.208,A -85,B 0,C 180,E1 10100.72,E2 10100.72} C_VEL
LIN {X 0,Y 322.712,Z 432.474,A -85,B 0,C 180,E1 10097.676,E2 10097.676} C_VEL
LIN {X 0,Y 318.611,Z 427.55,A -85,B 0,C 180,E1 10094.726,E2 10094.726} C_VEL
LIN {X 0,Y 315.26,Z 422.759,A -85,B 0,C 180,E1 10091.618,E2 10091.618} C_VEL
LIN {X 0,Y 313.766,Z 420.728,A -85,B 0,C 180,E1 10089.909,E2 10089.909} C_VEL
LIN {X 0,Y 311.805,Z 417.051,A -85,B 0,C 180,E1 10086.814,E2 10086.814} C_VEL
LIN {X 0,Y 309.993,Z 415.106,A -85,B 0,C 180,E1 10080.739,E2 10080.739} C_VEL
LIN {X 0,Y 310.477,Z 415.886,A -85,B 0,C 180,E1 10076.677,E2 10076.677} C_VEL
LIN {X 0,Y 312.043,Z 417.394,A -85,B 0,C 180,E1 10073.191,E2 10073.191} C_VEL
LIN {X 0,Y 314.592,Z 421.727,A -85,B 0,C 180,E1 10069.563,E2 10069.563} C_VEL
LIN {X 0,Y 318.413,Z 427.856,A -85,B 0,C 180,E1 10065.822,E2 10065.822} C_VEL
LIN {X 0,Y 321.563,Z 433.085,A -85,B 0,C 180,E1 10063.378,E2 10063.378} C_VEL
LIN {X 0,Y 325.61,Z 439.819,A -85,B 0,C 180,E1 10060.725,E2 10060.725} C_VEL
LIN {X 0,Y 328.704,Z 446.274,A -85,B 0,C 180,E1 10058.872,E2 10058.872} C_VEL
LIN {X 0,Y 330.14,Z 449.928,A -85,B 0,C 180,E1 10058.036,E2 10058.036} C_VEL
LIN {X 0,Y 320.65,Z 561.641,A -85,B 0,C 180,E1 10055.808,E2 10055.808} C_VEL
LIN {X 0,Y 319.6,Z 569.338,A -85,B 0,C 180,E1 10055.821,E2 10055.821} C_VEL
LIN {X 0,Y 315.258,Z 589.856,A -85,B 0,C 180,E1 10056.439,E2 10056.439} C_VEL
LIN {X 0,Y 314.244,Z 596.436,A -85,B 0,C 180,E1 10056.411,E2 10056.411} C_VEL
LIN {X 0,Y 310.717,Z 619.788,A -85,B 0,C 180,E1 10055.804,E2 10055.804} C_VEL
LIN {X 0,Y 306.376,Z 639.344,A -85,B 0,C 180,E1 10055.125,E2 10055.125} C_VEL
LIN {X 0,Y 301.496,Z 657.213,A -85,B 0,C 180,E1 10054.314,E2 10054.314} C_VEL
LIN {X 0,Y 294.804,Z 677.735,A -85,B 0,C 180,E1 10053.122,E2 10053.122} C_VEL
LIN {X 0,Y 287.32,Z 696.716,A -85,B 0,C 180,E1 10051.691,E2 10051.691} C_VEL
LIN {X 0,Y 280.444,Z 712.193,A -85,B 0,C 180,E1 10050.261,E2 10050.261} C_VEL
LIN {X 0,Y 271.637,Z 730.079,A -85,B 0,C 180,E1 10048.239,E2 10048.239} C_VEL
LIN {X 0,Y 261.955,Z 747.392,A -85,B 0,C 180,E1 10045.757,E2 10045.757} C_VEL
LIN {X 0,Y 253.651,Z 761.129,A -85,B 0,C 180,E1 10043.336,E2 10043.336} C_VEL
LIN {X 0,Y 243.874,Z 776.311,A -85,B 0,C 180,E1 10040.055,E2 10040.055} C_VEL
LIN {X 0,Y 234.421,Z 789.908,A -85,B 0,C 180,E1 10036.294,E2 10036.294} C_VEL
LIN {X 0,Y 226.932,Z 800.4,A -85,B 0,C 180,E1 10032.727,E2 10032.727} C_VEL
LIN {X 0,Y 218.576,Z 812.031,A -85,B 0,C 180,E1 10027.803,E2 10027.803} C_VEL
LIN {X 0,Y 212.079,Z 821.109,A -85,B 0,C 180,E1 10022.831,E2 10022.831} C_VEL
LIN {X 0,Y 207.286,Z 828.308,A -85,B 0,C 180,E1 10017.896,E2 10017.896} C_VEL
LIN {X 0,Y 203.123,Z 835.449,A -85,B 0,C 180,E1 10011.513,E2 10011.513} C_VEL
LIN {X 0,Y 201.038,Z 839.987,A -85,B 0,C 180,E1 10005.875,E2 10005.875} C_VEL
LIN {X 0,Y 200.199,Z 842.836,A -85,B 0,C 180,E1 10000.94,E2 10000.94} C_VEL
LIN {X 0,Y 199.985,Z 844.647,A -85,B 0,C 180,E1 9996.027,E2 9996.027} C_VEL
LIN {X 0,Y 200.006,Z 845.432,A -85,B 0,C 180,E1 9991.076,E2 9991.076} C_VEL
LIN {X 0,Y 199.982,Z 845.142,A -85,B 0,C 180,E1 9985.986,E2 9985.986} C_VEL
LIN {X 0,Y 200.103,Z 843.395,A -85,B 0,C 180,E1 9980.219,E2 9980.219} C_VEL
LIN {X 0,Y 200.896,Z 840.38,A -85,B 0,C 180,E1 9974.706,E2 9974.706} C_VEL
LIN {X 0,Y 202.647,Z 836.336,A -85,B 0,C 180,E1 9969.494,E2 9969.494} C_VEL
LIN {X 0,Y 206.197,Z 830.149,A -85,B 0,C 180,E1 9963.506,E2 9963.506} C_VEL
LIN {X 0,Y 211.481,Z 821.978,A -85,B 0,C 180,E1 9957.708,E2 9957.708} C_VEL
LIN {X 0,Y 217.087,Z 814.029,A -85,B 0,C 180,E1 9953.221,E2 9953.221} C_VEL
LIN {X 0,Y 225.141,Z 802.963,A -85,B 0,C 180,E1 9948.231,E2 9948.231} C_VEL
LIN {X 0,Y 233.665,Z 790.979,A -85,B 0,C 180,E1 9944.04,E2 9944.04} C_VEL
LIN {X 0,Y 241.625,Z 779.525,A -85,B 0,C 180,E1 9940.778,E2 9940.778} C_VEL
LIN {X 0,Y 251.822,Z 764.1,A -85,B 0,C 180,E1 9937.24,E2 9937.24} C_VEL
LIN {X 0,Y 260.923,Z 749.144,A -85,B 0,C 180,E1 9934.527,E2 9934.527} C_VEL
LIN {X 0,Y 269.329,Z 734.265,A -85,B 0,C 180,E1 9932.316,E2 9932.316} C_VEL
LIN {X 0,Y 279.338,Z 714.583,A -85,B 0,C 180,E1 9929.982,E2 9929.982} C_VEL
LIN {X 0,Y 286.801,Z 697.933,A -85,B 0,C 180,E1 9928.412,E2 9928.412} C_VEL
LIN {X 0,Y 294.04,Z 679.709,A -85,B 0,C 180,E1 9927.015,E2 9927.015} C_VEL
LIN {X 0,Y 301.11,Z 658.531,A -85,B 0,C 180,E1 9925.752,E2 9925.752} C_VEL
LIN {X 0,Y 306.065,Z 640.574,A -85,B 0,C 180,E1 9924.924,E2 9924.924} C_VEL
LIN {X 0,Y 310.592,Z 620.385,A -85,B 0,C 180,E1 9924.215,E2 9924.215} C_VEL
LIN {X 0,Y 314.107,Z 597.422,A -85,B 0,C 180,E1 9923.613,E2 9923.613} C_VEL
LIN {X 0,Y 326.83,Z 453.957,A -85,B 0,C 180,E1 9920.739,E2 9920.739} C_VEL
LIN {X 0,Y 323.628,Z 446.959,A -85,B 0,C 180,E1 9918.742,E2 9918.742} C_VEL
LIN {X 0,Y 319.606,Z 440.039,A -85,B 0,C 180,E1 9915.98,E2 9915.98} C_VEL
LIN {X 0,Y 316.119,Z 434.049,A -85,B 0,C 180,E1 9913.07,E2 9913.07} C_VEL
LIN {X 0,Y 313.296,Z 429.436,A -85,B 0,C 180,E1 9910.109,E2 9910.109} C_VEL
LIN {X 0,Y 310.662,Z 424.902,A -85,B 0,C 180,E1 9906.097,E2 9906.097} C_VEL
LIN {X 0,Y 309.013,Z 423.04,A -85,B 0,C 180,E1 9900.185,E2 9900.185} C_VEL
LIN {X 0,Y 309.537,Z 423.885,A -85,B 0,C 180,E1 9896.11,E2 9896.11} C_VEL
LIN {X 0,Y 310.966,Z 425.377,A -85,B 0,C 180,E1 9892.889,E2 9892.889} C_VEL
LIN {X 0,Y 313.942,Z 430.469,A -85,B 0,C 180,E1 9888.705,E2 9888.705} C_VEL
LIN {X 0,Y 317.311,Z 435.353,A -85,B 0,C 180,E1 9885.492,E2 9885.492} C_VEL
LIN {X 0,Y 322.87,Z 441.603,A -85,B 0,C 180,E1 9881.587,E2 9881.587} C_VEL
LIN {X 0,Y 327.668,Z 445.035,A -85,B 0,C 180,E1 9878.708,E2 9878.708} C_VEL
LIN {X 0,Y 331.76,Z 448.833,A -85,B 0,C 180,E1 9875.992,E2 9875.992} C_VEL
LIN {X 0,Y 335.368,Z 451.434,A -85,B 0,C 180,E1 9873.244,E2 9873.244} C_VEL
LIN {X 0,Y 337.795,Z 452.989,A -85,B 0,C 180,E1 9871.25,E2 9871.25} C_VEL
LIN {X 0,Y 340.521,Z 456.333,A -85,B 0,C 180,E1 9868.49,E2 9868.49} C_VEL
LIN {X 0,Y 343.802,Z 459.057,A -85,B 0,C 180,E1 9865.046,E2 9865.046} C_VEL
LIN {X 0,Y 345.437,Z 460.201,A -85,B 0,C 180,E1 9863.397,E2 9863.397} C_VEL
LIN {X 0,Y 348.219,Z 463.798,A -85,B 0,C 180,E1 9860.185,E2 9860.185} C_VEL
LIN {X 0,Y 350.968,Z 466.032,A -85,B 0,C 180,E1 9857.066,E2 9857.066} C_VEL
LIN {X 0,Y 352.957,Z 467.324,A -85,B 0,C 180,E1 9854.796,E2 9854.796} C_VEL
LIN {X 0,Y 355.13,Z 470.296,A -85,B 0,C 180,E1 9851.988,E2 9851.988} C_VEL
LIN {X 0,Y 357.489,Z 472.486,A -85,B 0,C 180,E1 9848.965,E2 9848.965} C_VEL
LIN {X 0,Y 360.3,Z 474.093,A -85,B 0,C 180,E1 9845.254,E2 9845.254} C_VEL
LIN {X 0,Y 361.139,Z 474.993,A -85,B 0,C 180,E1 9844.004,E2 9844.004} C_VEL
LIN {X 0,Y 363.352,Z 478.053,A -85,B 0,C 180,E1 9840.418,E2 9840.418} C_VEL
LIN {X 0,Y 365.218,Z 479.749,A -85,B 0,C 180,E1 9837.206,E2 9837.206} C_VEL
LIN {X 0,Y 367.18,Z 480.902,A -85,B 0,C 180,E1 9833.766,E2 9833.766} C_VEL
LIN {X 0,Y 368.795,Z 481.681,A -85,B 0,C 180,E1 9830.273,E2 9830.273} C_VEL
LIN {X 0,Y 369.741,Z 483.028,A -85,B 0,C 180,E1 9827.792,E2 9827.792} C_VEL
LIN {X 0,Y 370.835,Z 484.741,A -85,B 0,C 180,E1 9824.521,E2 9824.521} C_VEL
LIN {X 0,Y 371.742,Z 485.839,A -85,B 0,C 180,E1 9820.972,E2 9820.972} C_VEL
LIN {X 0,Y 372.386,Z 486.497,A -85,B 0,C 180,E1 9817.793,E2 9817.793} C_VEL
LIN {X 0,Y 372.874,Z 486.915,A -85,B 0,C 180,E1 9813.998,E2 9813.998} C_VEL
LIN {X 0,Y 373.046,Z 487.009,A -85,B 0,C 180,E1 9810.768,E2 9810.768} C_VEL
LIN {X 0,Y 372.952,Z 486.931,A -85,B 0,C 180,E1 9806.926,E2 9806.926} C_VEL
LIN {X 0,Y 372.624,Z 486.713,A -85,B 0,C 180,E1 9803.839,E2 9803.839} C_VEL
LIN {X 0,Y 372.055,Z 486.146,A -85,B 0,C 180,E1 9800.253,E2 9800.253} C_VEL
LIN {X 0,Y 371.201,Z 485.238,A -85,B 0,C 180,E1 9796.923,E2 9796.923} C_VEL
LIN {X 0,Y 370.249,Z 483.775,A -85,B 0,C 180,E1 9793.471,E2 9793.471} C_VEL
LIN {X 0,Y 368.961,Z 481.819,A -85,B 0,C 180,E1 9790.109,E2 9790.109} C_VEL
LIN {X 0,Y 367.554,Z 481.097,A -85,B 0,C 180,E1 9787.108,E2 9787.108} C_VEL
LIN {X 0,Y 365.562,Z 479.973,A -85,B 0,C 180,E1 9783.349,E2 9783.349} C_VEL
LIN {X 0,Y 363.755,Z 478.471,A -85,B 0,C 180,E1 9780.295,E2 9780.295} C_VEL
LIN {X 0,Y 362,Z 476.33,A -85,B 0,C 180,E1 9777.396,E2 9777.396} C_VEL
LIN {X 0,Y 360.416,Z 474.152,A -85,B 0,C 180,E1 9774.923,E2 9774.923} C_VEL
LIN {X 0,Y 357.655,Z 472.595,A -85,B 0,C 180,E1 9771.23,E2 9771.23} C_VEL
LIN {X 0,Y 355.249,Z 470.426,A -85,B 0,C 180,E1 9768.162,E2 9768.162} C_VEL
LIN {X 0,Y 353.032,Z 467.456,A -85,B 0,C 180,E1 9765.307,E2 9765.307} C_VEL
LIN {X 0,Y 351.868,Z 466.512,A -85,B 0,C 180,E1 9763.895,E2 9763.895} C_VEL
LIN {X 0,Y 349.049,Z 464.573,A -85,B 0,C 180,E1 9760.776,E2 9760.776} C_VEL
LIN {X 0,Y 346.51,Z 461.893,A -85,B 0,C 180,E1 9757.924,E2 9757.924} C_VEL
LIN {X 0,Y 344.839,Z 459.602,A -85,B 0,C 180,E1 9756.008,E2 9756.008} C_VEL
LIN {X 0,Y 341.845,Z 457.613,A -85,B 0,C 180,E1 9752.958,E2 9752.958} C_VEL
LIN {X 0,Y 338.875,Z 454.493,A -85,B 0,C 180,E1 9749.839,E2 9749.839} C_VEL
LIN {X 0,Y 337.113,Z 452.354,A -85,B 0,C 180,E1 9748.137,E2 9748.137} C_VEL
LIN {X 0,Y 333.347,Z 450.127,A -85,B 0,C 180,E1 9745.209,E2 9745.209} C_VEL
LIN {X 0,Y 329.494,Z 446.885,A -85,B 0,C 180,E1 9742.479,E2 9742.479} C_VEL
LIN {X 0,Y 326.343,Z 443.938,A -85,B 0,C 180,E1 9740.443,E2 9740.443} C_VEL
LIN {X 0,Y 320.953,Z 439.9,A -85,B 0,C 180,E1 9737.215,E2 9737.215} C_VEL
LIN {X 0,Y 317.091,Z 435.134,A -85,B 0,C 180,E1 9734.331,E2 9734.331} C_VEL
LIN {X 0,Y 313.792,Z 430.136,A -85,B 0,C 180,E1 9731.115,E2 9731.115} C_VEL
LIN {X 0,Y 310.729,Z 424.943,A -85,B 0,C 180,E1 9726.652,E2 9726.652} C_VEL
LIN {X 0,Y 309.018,Z 423.046,A -85,B 0,C 180,E1 9720.742,E2 9720.742} C_VEL
LIN {X 0,Y 309.502,Z 423.845,A -85,B 0,C 180,E1 9716.666,E2 9716.666} C_VEL
LIN {X 0,Y 310.952,Z 425.351,A -85,B 0,C 180,E1 9713.353,E2 9713.353} C_VEL
LIN {X 0,Y 313.916,Z 430.449,A -85,B 0,C 180,E1 9709.169,E2 9709.169} C_VEL
LIN {X 0,Y 317.1,Z 435.77,A -85,B 0,C 180,E1 9706.042,E2 9706.042} C_VEL
LIN {X 0,Y 321.058,Z 442.367,A -85,B 0,C 180,E1 9702.978,E2 9702.978} C_VEL
LIN {X 0,Y 324.703,Z 449.088,A -85,B 0,C 180,E1 9700.576,E2 9700.576} C_VEL
LIN {X 0,Y 326.81,Z 454.283,A -85,B 0,C 180,E1 9699.251,E2 9699.251} C_VEL
LIN {X 0,Y 314.244,Z 596.436,A -85,B 0,C 180,E1 9696.411,E2 9696.411} C_VEL
LIN {X 0,Y 312.6,Z 605.149,A -85,B 0,C 180,E1 9696.426,E2 9696.426} C_VEL
LIN {X 0,Y 307.429,Z 622.124,A -85,B 0,C 180,E1 9696.889,E2 9696.889} C_VEL
LIN {X 0,Y 305.388,Z 629.622,A -85,B 0,C 180,E1 9696.845,E2 9696.845} C_VEL
LIN {X 0,Y 305.153,Z 630.696,A -85,B 0,C 180,E1 9696.814,E2 9696.814} C_VEL
LIN {X 0,Y 299.52,Z 652.226,A -85,B 0,C 180,E1 9695.943,E2 9695.943} C_VEL
LIN {X 0,Y 293.945,Z 669.645,A -85,B 0,C 180,E1 9695.023,E2 9695.023} C_VEL
LIN {X 0,Y 286.985,Z 688.338,A -85,B 0,C 180,E1 9693.78,E2 9693.78} C_VEL
LIN {X 0,Y 278.306,Z 708.168,A -85,B 0,C 180,E1 9692.1,E2 9692.1} C_VEL
LIN {X 0,Y 270.267,Z 724.324,A -85,B 0,C 180,E1 9690.385,E2 9690.385} C_VEL
LIN {X 0,Y 261.345,Z 740.572,A -85,B 0,C 180,E1 9688.273,E2 9688.273} C_VEL
LIN {X 0,Y 251.088,Z 757.392,A -85,B 0,C 180,E1 9685.515,E2 9685.515} C_VEL
LIN {X 0,Y 242.263,Z 770.717,A -85,B 0,C 180,E1 9682.799,E2 9682.799} C_VEL
LIN {X 0,Y 233.457,Z 783.283,A -85,B 0,C 180,E1 9679.669,E2 9679.669} C_VEL
LIN {X 0,Y 223.221,Z 797.112,A -85,B 0,C 180,E1 9675.313,E2 9675.313} C_VEL
LIN {X 0,Y 215.427,Z 807.322,A -85,B 0,C 180,E1 9671.227,E2 9671.227} C_VEL
LIN {X 0,Y 208.256,Z 816.768,A -85,B 0,C 180,E1 9666.535,E2 9666.535} C_VEL
LIN {X 0,Y 201.578,Z 825.819,A -85,B 0,C 180,E1 9660.723,E2 9660.723} C_VEL
LIN {X 0,Y 197.336,Z 832.08,A -85,B 0,C 180,E1 9655.51,E2 9655.51} C_VEL
LIN {X 0,Y 194.433,Z 837.095,A -85,B 0,C 180,E1 9650.153,E2 9650.153} C_VEL
LIN {X 0,Y 192.527,Z 841.601,A -85,B 0,C 180,E1 9643.515,E2 9643.515} C_VEL
LIN {X 0,Y 192.017,Z 843.975,A -85,B 0,C 180,E1 9637.781,E2 9637.781} C_VEL
LIN {X 0,Y 191.993,Z 845.008,A -85,B 0,C 180,E1 9632.985,E2 9632.985} C_VEL
LIN {X 0,Y 192.006,Z 845.149,A -85,B 0,C 180,E1 9628.508,E2 9628.508} C_VEL
LIN {X 0,Y 191.988,Z 844.397,A -85,B 0,C 180,E1 9623.721,E2 9623.721} C_VEL
LIN {X 0,Y 192.242,Z 842.584,A -85,B 0,C 180,E1 9618.601,E2 9618.601} C_VEL
LIN {X 0,Y 193.19,Z 839.734,A -85,B 0,C 180,E1 9613.462,E2 9613.462} C_VEL
LIN {X 0,Y 195.411,Z 835.32,A -85,B 0,C 180,E1 9607.752,E2 9607.752} C_VEL
LIN {X 0,Y 199.969,Z 828.117,A -85,B 0,C 180,E1 9601.046,E2 9601.046} C_VEL
LIN {X 0,Y 205.096,Z 820.942,A -85,B 0,C 180,E1 9595.972,E2 9595.972} C_VEL
LIN {X 0,Y 212.081,Z 811.773,A -85,B 0,C 180,E1 9590.822,E2 9590.822} C_VEL
LIN {X 0,Y 220.915,Z 800.142,A -85,B 0,C 180,E1 9585.815,E2 9585.815} C_VEL
LIN {X 0,Y 229.051,Z 789.284,A -85,B 0,C 180,E1 9582.092,E2 9582.092} C_VEL
LIN {X 0,Y 239.251,Z 775.188,A -85,B 0,C 180,E1 9578.219,E2 9578.219} C_VEL
LIN {X 0,Y 249.148,Z 760.376,A -85,B 0,C 180,E1 9575.05,E2 9575.05} C_VEL
LIN {X 0,Y 257.919,Z 746.335,A -85,B 0,C 180,E1 9572.605,E2 9572.605} C_VEL
LIN {X 0,Y 268.133,Z 728.45,A -85,B 0,C 180,E1 9570.106,E2 9570.106} C_VEL
LIN {X 0,Y 276.467,Z 712.002,A -85,B 0,C 180,E1 9568.279,E2 9568.279} C_VEL
LIN {X 0,Y 283.562,Z 696.469,A -85,B 0,C 180,E1 9566.865,E2 9566.865} C_VEL
LIN {X 0,Y 291.508,Z 676.76,A -85,B 0,C 180,E1 9565.411,E2 9565.411} C_VEL
LIN {X 0,Y 298.09,Z 656.971,A -85,B 0,C 180,E1 9564.289,E2 9564.289} C_VEL
LIN {X 0,Y 303.081,Z 639.105,A -85,B 0,C 180,E1 9563.496,E2 9563.496} C_VEL
LIN {X 0,Y 308.004,Z 617.07,A -85,B 0,C 180,E1 9562.758,E2 9562.758} C_VEL
LIN {X 0,Y 311.178,Z 595.378,A -85,B 0,C 180,E1 9562.217,E2 9562.217} C_VEL
LIN {X 0,Y 323.622,Z 458.429,A -85,B 0,C 180,E1 9559.492,E2 9559.492} C_VEL
LIN {X 0,Y 321.166,Z 453.095,A -85,B 0,C 180,E1 9557.857,E2 9557.857} C_VEL
LIN {X 0,Y 316.725,Z 445.214,A -85,B 0,C 180,E1 9554.535,E2 9554.535} C_VEL
LIN {X 0,Y 314.178,Z 440.96,A -85,B 0,C 180,E1 9552.218,E2 9552.218} C_VEL
LIN {X 0,Y 312.011,Z 437.147,A -85,B 0,C 180,E1 9549.779,E2 9549.779} C_VEL
LIN {X 0,Y 309.59,Z 432.793,A -85,B 0,C 180,E1 9545.932,E2 9545.932} C_VEL
LIN {X 0,Y 308.039,Z 430.98,A -85,B 0,C 180,E1 9540.186,E2 9540.186} C_VEL
LIN {X 0,Y 308.562,Z 431.847,A -85,B 0,C 180,E1 9536.098,E2 9536.098} C_VEL
LIN {X 0,Y 309.836,Z 433.199,A -85,B 0,C 180,E1 9533.142,E2 9533.142} C_VEL
LIN {X 0,Y 312.635,Z 438.176,A -85,B 0,C 180,E1 9529.03,E2 9529.03} C_VEL
LIN {X 0,Y 316.015,Z 443.155,A -85,B 0,C 180,E1 9525.712,E2 9525.712} C_VEL
LIN {X 0,Y 321.213,Z 449.182,A -85,B 0,C 180,E1 9521.958,E2 9521.958} C_VEL
LIN {X 0,Y 326.313,Z 452.884,A -85,B 0,C 180,E1 9518.898,E2 9518.898} C_VEL
LIN {X 0,Y 330.039,Z 456.348,A -85,B 0,C 180,E1 9516.428,E2 9516.428} C_VEL
LIN {X 0,Y 334.028,Z 459.214,A -85,B 0,C 180,E1 9513.506,E2 9513.506} C_VEL
LIN {X 0,Y 336.568,Z 460.858,A -85,B 0,C 180,E1 9511.426,E2 9511.426} C_VEL
LIN {X 0,Y 339.43,Z 464.263,A -85,B 0,C 180,E1 9508.575,E2 9508.575} C_VEL
LIN {X 0,Y 342.905,Z 467.073,A -85,B 0,C 180,E1 9504.941,E2 9504.941} C_VEL
LIN {X 0,Y 344.265,Z 468.078,A -85,B 0,C 180,E1 9503.56,E2 9503.56} C_VEL
LIN {X 0,Y 347.168,Z 471.734,A -85,B 0,C 180,E1 9500.255,E2 9500.255} C_VEL
LIN {X 0,Y 350.076,Z 474.048,A -85,B 0,C 180,E1 9496.952,E2 9496.952} C_VEL
LIN {X 0,Y 351.836,Z 475.197,A -85,B 0,C 180,E1 9494.959,E2 9494.959} C_VEL
LIN {X 0,Y 354.129,Z 478.284,A -85,B 0,C 180,E1 9492,E2 9492} C_VEL
LIN {X 0,Y 356.546,Z 480.475,A -85,B 0,C 180,E1 9488.913,E2 9488.913} C_VEL
LIN {X 0,Y 359.404,Z 482.083,A -85,B 0,C 180,E1 9485.125,E2 9485.125} C_VEL
LIN {X 0,Y 361.457,Z 484.958,A -85,B 0,C 180,E1 9481.873,E2 9481.873} C_VEL
LIN {X 0,Y 363.635,Z 487.203,A -85,B 0,C 180,E1 9478.373,E2 9478.373} C_VEL
LIN {X 0,Y 365.512,Z 488.521,A -85,B 0,C 180,E1 9474.914,E2 9474.914} C_VEL
LIN {X 0,Y 367.386,Z 489.358,A -85,B 0,C 180,E1 9471.388,E2 9471.388} C_VEL
LIN {X 0,Y 368.555,Z 490.502,A -85,B 0,C 180,E1 9468.506,E2 9468.506} C_VEL
LIN {X 0,Y 369.552,Z 492.296,A -85,B 0,C 180,E1 9465.375,E2 9465.375} C_VEL
LIN {X 0,Y 370.633,Z 493.591,A -85,B 0,C 180,E1 9461.831,E2 9461.831} C_VEL
LIN {X 0,Y 371.298,Z 494.343,A -85,B 0,C 180,E1 9458.361,E2 9458.361} C_VEL
LIN {X 0,Y 371.861,Z 494.75,A -85,B 0,C 180,E1 9454.936,E2 9454.936} C_VEL
LIN {X 0,Y 372.048,Z 494.941,A -85,B 0,C 180,E1 9451.34,E2 9451.34} C_VEL
LIN {X 0,Y 372.055,Z 494.957,A -85,B 0,C 180,E1 9448.152,E2 9448.152} C_VEL
LIN {X 0,Y 371.732,Z 494.706,A -85,B 0,C 180,E1 9444.443,E2 9444.443} C_VEL
LIN {X 0,Y 371.247,Z 494.259,A -85,B 0,C 180,E1 9441.271,E2 9441.271} C_VEL
LIN {X 0,Y 370.401,Z 493.412,A -85,B 0,C 180,E1 9437.529,E2 9437.529} C_VEL
LIN {X 0,Y 369.497,Z 492.198,A -85,B 0,C 180,E1 9434.436,E2 9434.436} C_VEL
LIN {X 0,Y 368.412,Z 490.214,A -85,B 0,C 180,E1 9430.994,E2 9430.994} C_VEL
LIN {X 0,Y 366.985,Z 489.199,A -85,B 0,C 180,E1 9427.916,E2 9427.916} C_VEL
LIN {X 0,Y 365.325,Z 488.423,A -85,B 0,C 180,E1 9424.726,E2 9424.726} C_VEL
LIN {X 0,Y 363.245,Z 486.868,A -85,B 0,C 180,E1 9421.024,E2 9421.024} C_VEL
LIN {X 0,Y 361.294,Z 484.744,A -85,B 0,C 180,E1 9417.869,E2 9417.869} C_VEL
LIN {X 0,Y 359.38,Z 482.07,A -85,B 0,C 180,E1 9414.838,E2 9414.838} C_VEL
LIN {X 0,Y 356.46,Z 480.417,A -85,B 0,C 180,E1 9410.984,E2 9410.984} C_VEL
LIN {X 0,Y 354.095,Z 478.246,A -85,B 0,C 180,E1 9407.956,E2 9407.956} C_VEL
LIN {X 0,Y 351.836,Z 475.197,A -85,B 0,C 180,E1 9405.041,E2 9405.041} C_VEL
LIN {X 0,Y 348.349,Z 472.795,A -85,B 0,C 180,E1 9401.094,E2 9401.094} C_VEL
LIN {X 0,Y 345.678,Z 470.166,A -85,B 0,C 180,E1 9398.119,E2 9398.119} C_VEL
LIN {X 0,Y 343.621,Z 467.449,A -85,B 0,C 180,E1 9395.793,E2 9395.793} C_VEL
LIN {X 0,Y 340.764,Z 465.536,A -85,B 0,C 180,E1 9392.876,E2 9392.876} C_VEL
LIN {X 0,Y 337.831,Z 462.534,A -85,B 0,C 180,E1 9389.816,E2 9389.816} C_VEL
LIN {X 0,Y 335.811,Z 460.151,A -85,B 0,C 180,E1 9387.869,E2 9387.869} C_VEL
LIN {X 0,Y 332.177,Z 458.036,A -85,B 0,C 180,E1 9385.113,E2 9385.113} C_VEL
LIN {X 0,Y 328.075,Z 454.599,A -85,B 0,C 180,E1 9382.204,E2 9382.204} C_VEL
LIN {X 0,Y 324.786,Z 451.625,A -85,B 0,C 180,E1 9380.129,E2 9380.129} C_VEL
LIN {X 0,Y 319.217,Z 447.321,A -85,B 0,C 180,E1 9376.748,E2 9376.748} C_VEL
LIN {X 0,Y 315.588,Z 442.714,A -85,B 0,C 180,E1 9373.933,E2 9373.933} C_VEL
LIN {X 0,Y 311.961,Z 437.073,A -85,B 0,C 180,E1 9370.153,E2 9370.153} C_VEL
LIN {X 0,Y 309.556,Z 432.768,A -85,B 0,C 180,E1 9366.305,E2 9366.305} C_VEL
LIN {X 0,Y 308.035,Z 430.99,A -85,B 0,C 180,E1 9360.558,E2 9360.558} C_VEL
LIN {X 0,Y 308.526,Z 431.806,A -85,B 0,C 180,E1 9356.656,E2 9356.656} C_VEL
LIN {X 0,Y 309.822,Z 433.171,A -85,B 0,C 180,E1 9353.608,E2 9353.608} C_VEL
LIN {X 0,Y 312.609,Z 438.154,A -85,B 0,C 180,E1 9349.496,E2 9349.496} C_VEL
LIN {X 0,Y 315.596,Z 443.315,A -85,B 0,C 180,E1 9346.441,E2 9346.441} C_VEL
LIN {X 0,Y 319.431,Z 449.979,A -85,B 0,C 180,E1 9343.357,E2 9343.357} C_VEL
LIN {X 0,Y 322.645,Z 456.119,A -85,B 0,C 180,E1 9341.152,E2 9341.152} C_VEL
LIN {X 0,Y 323.625,Z 458.697,A -85,B 0,C 180,E1 9340.489,E2 9340.489} C_VEL
LIN {X 0,Y 310.89,Z 598.126,A -85,B 0,C 180,E1 9337.724,E2 9337.724} C_VEL
LIN {X 0,Y 306.881,Z 622.495,A -85,B 0,C 180,E1 9337.079,E2 9337.079} C_VEL
LIN {X 0,Y 305.153,Z 630.696,A -85,B 0,C 180,E1 9336.814,E2 9336.814} C_VEL
LIN {X 0,Y 303.072,Z 638.172,A -85,B 0,C 180,E1 9336.724,E2 9336.724} C_VEL
LIN {X 0,Y 295.428,Z 656.74,A -85,B 0,C 180,E1 9336.979,E2 9336.979} C_VEL
LIN {X 0,Y 292.592,Z 663.878,A -85,B 0,C 180,E1 9336.781,E2 9336.781} C_VEL
LIN {X 0,Y 285.462,Z 683.157,A -85,B 0,C 180,E1 9335.595,E2 9335.595} C_VEL
LIN {X 0,Y 278.05,Z 700.564,A -85,B 0,C 180,E1 9334.259,E2 9334.259} C_VEL
LIN {X 0,Y 268.186,Z 720.636,A -85,B 0,C 180,E1 9332.304,E2 9332.304} C_VEL
LIN {X 0,Y 259.396,Z 736.412,A -85,B 0,C 180,E1 9330.363,E2 9330.363} C_VEL
LIN {X 0,Y 249.919,Z 751.955,A -85,B 0,C 180,E1 9328.009,E2 9328.009} C_VEL
LIN {X 0,Y 239.28,Z 767.778,A -85,B 0,C 180,E1 9324.983,E2 9324.983} C_VEL
LIN {X 0,Y 229.968,Z 780.617,A -85,B 0,C 180,E1 9321.9,E2 9321.9} C_VEL
LIN {X 0,Y 220.828,Z 792.621,A -85,B 0,C 180,E1 9318.336,E2 9318.336} C_VEL
LIN {X 0,Y 210.652,Z 805.36,A -85,B 0,C 180,E1 9313.49,E2 9313.49} C_VEL
LIN {X 0,Y 203.074,Z 814.7,A -85,B 0,C 180,E1 9308.929,E2 9308.929} C_VEL
LIN {X 0,Y 196.034,Z 823.635,A -85,B 0,C 180,E1 9303.424,E2 9303.424} C_VEL
LIN {X 0,Y 190.365,Z 831.2,A -85,B 0,C 180,E1 9297.19,E2 9297.19} C_VEL
LIN {X 0,Y 187.031,Z 836.333,A -85,B 0,C 180,E1 9291.645,E2 9291.645} C_VEL
LIN {X 0,Y 184.948,Z 840.462,A -85,B 0,C 180,E1 9285.682,E2 9285.682} C_VEL
LIN {X 0,Y 184.051,Z 843.555,A -85,B 0,C 180,E1 9278.749,E2 9278.749} C_VEL
LIN {X 0,Y 183.992,Z 844.731,A -85,B 0,C 180,E1 9273.427,E2 9273.427} C_VEL
LIN {X 0,Y 184.011,Z 844.928,A -85,B 0,C 180,E1 9268.755,E2 9268.755} C_VEL
LIN {X 0,Y 183.99,Z 844.231,A -85,B 0,C 180,E1 9263.761,E2 9263.761} C_VEL
LIN {X 0,Y 184.257,Z 842.472,A -85,B 0,C 180,E1 9258.418,E2 9258.418} C_VEL
LIN {X 0,Y 185.274,Z 839.676,A -85,B 0,C 180,E1 9253.058,E2 9253.058} C_VEL
LIN {X 0,Y 187.49,Z 835.572,A -85,B 0,C 180,E1 9247.421,E2 9247.421} C_VEL
LIN {X 0,Y 192.035,Z 828.91,A -85,B 0,C 180,E1 9240.698,E2 9240.698} C_VEL
LIN {X 0,Y 197.665,Z 821.463,A -85,B 0,C 180,E1 9235.14,E2 9235.14} C_VEL
LIN {X 0,Y 204.037,Z 813.513,A -85,B 0,C 180,E1 9230.429,E2 9230.429} C_VEL
LIN {X 0,Y 213.062,Z 802.448,A -85,B 0,C 180,E1 9225.259,E2 9225.259} C_VEL
LIN {X 0,Y 222.471,Z 790.464,A -85,B 0,C 180,E1 9220.972,E2 9220.972} C_VEL
LIN {X 0,Y 231.169,Z 779.012,A -85,B 0,C 180,E1 9217.675,E2 9217.675} C_VEL
LIN {X 0,Y 242.116,Z 763.744,A -85,B 0,C 180,E1 9214.169,E2 9214.169} C_VEL
LIN {X 0,Y 251.985,Z 748.636,A -85,B 0,C 180,E1 9211.452,E2 9211.452} C_VEL
LIN {X 0,Y 260.846,Z 733.949,A -85,B 0,C 180,E1 9209.307,E2 9209.307} C_VEL
LIN {X 0,Y 271.158,Z 714.92,A -85,B 0,C 180,E1 9207.086,E2 9207.086} C_VEL
LIN {X 0,Y 279.211,Z 697.959,A -85,B 0,C 180,E1 9205.526,E2 9205.526} C_VEL
LIN {X 0,Y 286.51,Z 680.552,A -85,B 0,C 180,E1 9204.227,E2 9204.227} C_VEL
LIN {X 0,Y 294.258,Z 658.706,A -85,B 0,C 180,E1 9202.956,E2 9202.956} C_VEL
LIN {X 0,Y 299.758,Z 639.648,A -85,B 0,C 180,E1 9202.116,E2 9202.116} C_VEL
LIN {X 0,Y 304.721,Z 618.217,A -85,B 0,C 180,E1 9201.405,E2 9201.405} C_VEL
LIN {X 0,Y 308.134,Z 595.963,A -85,B 0,C 180,E1 9200.852,E2 9200.852} C_VEL
LIN {X 0,Y 320.559,Z 462.997,A -85,B 0,C 180,E1 9198.221,E2 9198.221} C_VEL
LIN {X 0,Y 317.36,Z 456.706,A -85,B 0,C 180,E1 9195.908,E2 9195.908} C_VEL
LIN {X 0,Y 313.38,Z 449.424,A -85,B 0,C 180,E1 9192.437,E2 9192.437} C_VEL
LIN {X 0,Y 310.736,Z 444.855,A -85,B 0,C 180,E1 9189.445,E2 9189.445} C_VEL
LIN {X 0,Y 308.521,Z 440.684,A -85,B 0,C 180,E1 9185.766,E2 9185.766} C_VEL
LIN {X 0,Y 307.064,Z 438.921,A -85,B 0,C 180,E1 9180.187,E2 9180.187} C_VEL
LIN {X 0,Y 307.586,Z 439.811,A -85,B 0,C 180,E1 9176.086,E2 9176.086} C_VEL
LIN {X 0,Y 308.712,Z 441.019,A -85,B 0,C 180,E1 9173.398,E2 9173.398} C_VEL
LIN {X 0,Y 311.339,Z 445.881,A -85,B 0,C 180,E1 9169.359,E2 9169.359} C_VEL
LIN {X 0,Y 314.725,Z 450.958,A -85,B 0,C 180,E1 9165.934,E2 9165.934} C_VEL
LIN {X 0,Y 319.571,Z 456.759,A -85,B 0,C 180,E1 9162.333,E2 9162.333} C_VEL
LIN {X 0,Y 324.834,Z 460.591,A -85,B 0,C 180,E1 9159.175,E2 9159.175} C_VEL
LIN {X 0,Y 328.713,Z 464.169,A -85,B 0,C 180,E1 9156.613,E2 9156.613} C_VEL
LIN {X 0,Y 332.702,Z 466.986,A -85,B 0,C 180,E1 9153.783,E2 9153.783} C_VEL
LIN {X 0,Y 335.27,Z 468.595,A -85,B 0,C 180,E1 9151.694,E2 9151.694} C_VEL
LIN {X 0,Y 338.166,Z 472.021,A -85,B 0,C 180,E1 9148.84,E2 9148.84} C_VEL
LIN {X 0,Y 341.837,Z 474.987,A -85,B 0,C 180,E1 9145.02,E2 9145.02} C_VEL
LIN {X 0,Y 343.085,Z 475.945,A -85,B 0,C 180,E1 9143.729,E2 9143.729} C_VEL
LIN {X 0,Y 345.988,Z 479.529,A -85,B 0,C 180,E1 9140.495,E2 9140.495} C_VEL
LIN {X 0,Y 348.879,Z 481.878,A -85,B 0,C 180,E1 9137.194,E2 9137.194} C_VEL
LIN {X 0,Y 350.722,Z 483.07,A -85,B 0,C 180,E1 9135.123,E2 9135.123} C_VEL
LIN {X 0,Y 353.064,Z 486.194,A -85,B 0,C 180,E1 9132.101,E2 9132.101} C_VEL
LIN {X 0,Y 355.443,Z 488.355,A -85,B 0,C 180,E1 9129.057,E2 9129.057} C_VEL
LIN {X 0,Y 358.323,Z 489.977,A -85,B 0,C 180,E1 9125.281,E2 9125.281} C_VEL
LIN {X 0,Y 360.445,Z 492.916,A -85,B 0,C 180,E1 9121.916,E2 9121.916} C_VEL
LIN {X 0,Y 362.633,Z 495.143,A -85,B 0,C 180,E1 9118.412,E2 9118.412} C_VEL
LIN {X 0,Y 364.496,Z 496.446,A -85,B 0,C 180,E1 9114.988,E2 9114.988} C_VEL
LIN {X 0,Y 366.37,Z 497.287,A -85,B 0,C 180,E1 9111.45,E2 9111.45} C_VEL
LIN {X 0,Y 367.562,Z 498.449,A -85,B 0,C 180,E1 9108.558,E2 9108.558} C_VEL
LIN {X 0,Y 368.561,Z 500.236,A -85,B 0,C 180,E1 9105.418,E2 9105.418} C_VEL
LIN {X 0,Y 369.585,Z 501.489,A -85,B 0,C 180,E1 9102.023,E2 9102.023} C_VEL
LIN {X 0,Y 370.296,Z 502.248,A -85,B 0,C 180,E1 9098.54,E2 9098.54} C_VEL
LIN {X 0,Y 370.815,Z 502.659,A -85,B 0,C 180,E1 9095.26,E2 9095.26} C_VEL
LIN {X 0,Y 371.072,Z 502.889,A -85,B 0,C 180,E1 9091.544,E2 9091.544} C_VEL
LIN {X 0,Y 371.072,Z 502.89,A -85,B 0,C 180,E1 9088.456,E2 9088.456} C_VEL
LIN {X 0,Y 370.815,Z 502.659,A -85,B 0,C 180,E1 9084.74,E2 9084.74} C_VEL
LIN {X 0,Y 370.296,Z 502.248,A -85,B 0,C 180,E1 9081.46,E2 9081.46} C_VEL
LIN {X 0,Y 369.524,Z 501.446,A -85,B 0,C 180,E1 9077.816,E2 9077.816} C_VEL
LIN {X 0,Y 368.561,Z 500.236,A -85,B 0,C 180,E1 9074.582,E2 9074.582} C_VEL
LIN {X 0,Y 367.48,Z 498.24,A -85,B 0,C 180,E1 9071.109,E2 9071.109} C_VEL
LIN {X 0,Y 366.069,Z 497.167,A -85,B 0,C 180,E1 9068.026,E2 9068.026} C_VEL
LIN {X 0,Y 364.312,Z 496.347,A -85,B 0,C 180,E1 9064.651,E2 9064.651} C_VEL
LIN {X 0,Y 362.202,Z 494.779,A -85,B 0,C 180,E1 9060.933,E2 9060.933} C_VEL
LIN {X 0,Y 360.269,Z 492.684,A -85,B 0,C 180,E1 9057.802,E2 9057.802} C_VEL
LIN {X 0,Y 358.324,Z 489.976,A -85,B 0,C 180,E1 9054.719,E2 9054.719} C_VEL
LIN {X 0,Y 355.434,Z 488.348,A -85,B 0,C 180,E1 9050.932,E2 9050.932} C_VEL
LIN {X 0,Y 353.064,Z 486.194,A -85,B 0,C 180,E1 9047.899,E2 9047.899} C_VEL
LIN {X 0,Y 350.646,Z 482.928,A -85,B 0,C 180,E1 9044.765,E2 9044.765} C_VEL
LIN {X 0,Y 347.293,Z 480.724,A -85,B 0,C 180,E1 9041.027,E2 9041.027} C_VEL
LIN {X 0,Y 344.543,Z 478.039,A -85,B 0,C 180,E1 9037.968,E2 9037.968} C_VEL
LIN {X 0,Y 342.364,Z 475.273,A -85,B 0,C 180,E1 9035.533,E2 9035.533} C_VEL
LIN {X 0,Y 339.513,Z 473.308,A -85,B 0,C 180,E1 9032.611,E2 9032.611} C_VEL
LIN {X 0,Y 336.51,Z 470.191,A -85,B 0,C 180,E1 9029.477,E2 9029.477} C_VEL
LIN {X 0,Y 334.663,Z 468.051,A -85,B 0,C 180,E1 9027.78,E2 9027.78} C_VEL
LIN {X 0,Y 331.009,Z 465.943,A -85,B 0,C 180,E1 9025.017,E2 9025.017} C_VEL
LIN {X 0,Y 326.86,Z 462.543,A -85,B 0,C 180,E1 9022.102,E2 9022.102} C_VEL
LIN {X 0,Y 323.315,Z 459.38,A -85,B 0,C 180,E1 9019.888,E2 9019.888} C_VEL
LIN {X 0,Y 317.625,Z 454.875,A -85,B 0,C 180,E1 9016.364,E2 9016.364} C_VEL
LIN {X 0,Y 314.202,Z 450.406,A -85,B 0,C 180,E1 9013.62,E2 9013.62} C_VEL
LIN {X 0,Y 310.689,Z 444.783,A -85,B 0,C 180,E1 9009.821,E2 9009.821} C_VEL
LIN {X 0,Y 308.488,Z 440.661,A -85,B 0,C 180,E1 9006.14,E2 9006.14} C_VEL
LIN {X 0,Y 307.06,Z 438.93,A -85,B 0,C 180,E1 9000.56,E2 9000.56} C_VEL
LIN {X 0,Y 307.55,Z 439.77,A -85,B 0,C 180,E1 8996.645,E2 8996.645} C_VEL
LIN {X 0,Y 308.738,Z 441.117,A -85,B 0,C 180,E1 8993.772,E2 8993.772} C_VEL
LIN {X 0,Y 311.383,Z 446.016,A -85,B 0,C 180,E1 8989.734,E2 8989.734} C_VEL
LIN {X 0,Y 314.203,Z 451.04,A -85,B 0,C 180,E1 8986.755,E2 8986.755} C_VEL
LIN {X 0,Y 317.761,Z 457.469,A -85,B 0,C 180,E1 8983.784,E2 8983.784} C_VEL
LIN {X 0,Y 320.594,Z 463.086,A -85,B 0,C 180,E1 8981.753,E2 8981.753} C_VEL
LIN {X 0,Y 307.921,Z 598.002,A -85,B 0,C 180,E1 8979.105,E2 8979.105} C_VEL
LIN {X 0,Y 303.857,Z 622.188,A -85,B 0,C 180,E1 8978.476,E2 8978.476} C_VEL
LIN {X 0,Y 299.355,Z 641.175,A -85,B 0,C 180,E1 8977.826,E2 8977.826} C_VEL
LIN {X 0,Y 293.451,Z 661.335,A -85,B 0,C 180,E1 8976.916,E2 8976.916} C_VEL
LIN {X 0,Y 292.592,Z 663.878,A -85,B 0,C 180,E1 8976.781,E2 8976.781} C_VEL
LIN {X 0,Y 289.623,Z 671.082,A -85,B 0,C 180,E1 8976.552,E2 8976.552} C_VEL
LIN {X 0,Y 280.208,Z 688.842,A -85,B 0,C 180,E1 8976.498,E2 8976.498} C_VEL
LIN {X 0,Y 276.82,Z 695.511,A -85,B 0,C 180,E1 8976.172,E2 8976.172} C_VEL
LIN {X 0,Y 268.738,Z 712.297,A -85,B 0,C 180,E1 8974.699,E2 8974.699} C_VEL
LIN {X 0,Y 258.821,Z 730.616,A -85,B 0,C 180,E1 8972.684,E2 8972.684} C_VEL
LIN {X 0,Y 248.505,Z 747.305,A -85,B 0,C 180,E1 8970.338,E2 8970.338} C_VEL
LIN {X 0,Y 239.31,Z 760.987,A -85,B 0,C 180,E1 8967.953,E2 8967.953} C_VEL
LIN {X 0,Y 228.126,Z 776.349,A -85,B 0,C 180,E1 8964.607,E2 8964.607} C_VEL
LIN {X 0,Y 218.302,Z 788.77,A -85,B 0,C 180,E1 8961.133,E2 8961.133} C_VEL
LIN {X 0,Y 209.343,Z 799.627,A -85,B 0,C 180,E1 8957.35,E2 8957.35} C_VEL
LIN {X 0,Y 199.495,Z 811.258,A -85,B 0,C 180,E1 8952.189,E2 8952.189} C_VEL
LIN {X 0,Y 191.656,Z 820.337,A -85,B 0,C 180,E1 8946.865,E2 8946.865} C_VEL
LIN {X 0,Y 185.711,Z 827.537,A -85,B 0,C 180,E1 8941.482,E2 8941.482} C_VEL
LIN {X 0,Y 180.464,Z 834.554,A -85,B 0,C 180,E1 8934.552,E2 8934.552} C_VEL
LIN {X 0,Y 177.567,Z 839.226,A -85,B 0,C 180,E1 8928.041,E2 8928.041} C_VEL
LIN {X 0,Y 176.313,Z 842.22,A -85,B 0,C 180,E1 8922.112,E2 8922.112} C_VEL
LIN {X 0,Y 175.991,Z 844.075,A -85,B 0,C 180,E1 8916.16,E2 8916.16} C_VEL
LIN {X 0,Y 176.025,Z 844.762,A -85,B 0,C 180,E1 8910.325,E2 8910.325} C_VEL
LIN {X 0,Y 175.986,Z 844.233,A -85,B 0,C 180,E1 8904.458,E2 8904.458} C_VEL
LIN {X 0,Y 176.275,Z 842.36,A -85,B 0,C 180,E1 8898.218,E2 8898.218} C_VEL
LIN {X 0,Y 177.502,Z 839.351,A -85,B 0,C 180,E1 8892.169,E2 8892.169} C_VEL
LIN {X 0,Y 180.095,Z 835.062,A -85,B 0,C 180,E1 8886.092,E2 8886.092} C_VEL
LIN {X 0,Y 185.424,Z 827.909,A -85,B 0,C 180,E1 8878.826,E2 8878.826} C_VEL
LIN {X 0,Y 191.286,Z 820.771,A -85,B 0,C 180,E1 8873.426,E2 8873.426} C_VEL
LIN {X 0,Y 198.593,Z 812.257,A -85,B 0,C 180,E1 8868.351,E2 8868.351} C_VEL
LIN {X 0,Y 208.817,Z 800.268,A -85,B 0,C 180,E1 8862.897,E2 8862.897} C_VEL
LIN {X 0,Y 217.715,Z 789.488,A -85,B 0,C 180,E1 8859.094,E2 8859.094} C_VEL
LIN {X 0,Y 227.485,Z 777.151,A -85,B 0,C 180,E1 8855.6,E2 8855.6} C_VEL
LIN {X 0,Y 238.71,Z 761.858,A -85,B 0,C 180,E1 8852.213,E2 8852.213} C_VEL
LIN {X 0,Y 248.164,Z 747.832,A -85,B 0,C 180,E1 8849.746,E2 8849.746} C_VEL
LIN {X 0,Y 257.694,Z 732.466,A -85,B 0,C 180,E1 8847.556,E2 8847.556} C_VEL
LIN {X 0,Y 267.965,Z 713.838,A -85,B 0,C 180,E1 8845.451,E2 8845.451} C_VEL
LIN {X 0,Y 276.21,Z 696.843,A -85,B 0,C 180,E1 8843.935,E2 8843.935} C_VEL
LIN {X 0,Y 283.839,Z 678.964,A -85,B 0,C 180,E1 8842.646,E2 8842.646} C_VEL
LIN {X 0,Y 291.494,Z 657.55,A -85,B 0,C 180,E1 8841.452,E2 8841.452} C_VEL
LIN {X 0,Y 297.035,Z 638.625,A -85,B 0,C 180,E1 8840.649,E2 8840.649} C_VEL
LIN {X 0,Y 302.162,Z 616.527,A -85,B 0,C 180,E1 8839.946,E2 8839.946} C_VEL
LIN {X 0,Y 305.464,Z 594.879,A -85,B 0,C 180,E1 8839.425,E2 8839.425} C_VEL
LIN {X 0,Y 317.62,Z 467.873,A -85,B 0,C 180,E1 8836.929,E2 8836.929} C_VEL
LIN {X 0,Y 313.69,Z 460.297,A -85,B 0,C 180,E1 8833.737,E2 8833.737} C_VEL
LIN {X 0,Y 311.321,Z 456.066,A -85,B 0,C 180,E1 8831.392,E2 8831.392} C_VEL
LIN {X 0,Y 309.473,Z 452.563,A -85,B 0,C 180,E1 8829.109,E2 8829.109} C_VEL
LIN {X 0,Y 307.362,Z 448.509,A -85,B 0,C 180,E1 8825.413,E2 8825.413} C_VEL
LIN {X 0,Y 306.083,Z 446.866,A -85,B 0,C 180,E1 8820,E2 8820} C_VEL
LIN {X 0,Y 306.667,Z 447.854,A -85,B 0,C 180,E1 8815.887,E2 8815.887} C_VEL
LIN {X 0,Y 307.633,Z 448.965,A -85,B 0,C 180,E1 8813.562,E2 8813.562} C_VEL
LIN {X 0,Y 310.121,Z 453.741,A -85,B 0,C 180,E1 8809.598,E2 8809.598} C_VEL
LIN {X 0,Y 314.57,Z 460.521,A -85,B 0,C 180,E1 8805.175,E2 8805.175} C_VEL
LIN {X 0,Y 319.315,Z 465.449,A -85,B 0,C 180,E1 8801.847,E2 8801.847} C_VEL
LIN {X 0,Y 323.494,Z 468.437,A -85,B 0,C 180,E1 8799.369,E2 8799.369} C_VEL
LIN {X 0,Y 327.518,Z 472.092,A -85,B 0,C 180,E1 8796.713,E2 8796.713} C_VEL
LIN {X 0,Y 331.56,Z 474.888,A -85,B 0,C 180,E1 8793.878,E2 8793.878} C_VEL
LIN {X 0,Y 334.161,Z 476.59,A -85,B 0,C 180,E1 8791.787,E2 8791.787} C_VEL
LIN {X 0,Y 337.084,Z 479.951,A -85,B 0,C 180,E1 8788.928,E2 8788.928} C_VEL
LIN {X 0,Y 340.778,Z 482.903,A -85,B 0,C 180,E1 8785.101,E2 8785.101} C_VEL
LIN {X 0,Y 342.007,Z 483.941,A -85,B 0,C 180,E1 8783.804,E2 8783.804} C_VEL
LIN {X 0,Y 345.056,Z 487.586,A -85,B 0,C 180,E1 8780.422,E2 8780.422} C_VEL
LIN {X 0,Y 347.992,Z 489.893,A -85,B 0,C 180,E1 8777.082,E2 8777.082} C_VEL
LIN {X 0,Y 349.612,Z 490.941,A -85,B 0,C 180,E1 8775.289,E2 8775.289} C_VEL
LIN {X 0,Y 352.093,Z 494.207,A -85,B 0,C 180,E1 8772.08,E2 8772.08} C_VEL
LIN {X 0,Y 354.534,Z 496.364,A -85,B 0,C 180,E1 8768.968,E2 8768.968} C_VEL
LIN {X 0,Y 357.404,Z 497.953,A -85,B 0,C 180,E1 8765.189,E2 8765.189} C_VEL
LIN {X 0,Y 359.47,Z 500.918,A -85,B 0,C 180,E1 8761.902,E2 8761.902} C_VEL
LIN {X 0,Y 361.659,Z 503.112,A -85,B 0,C 180,E1 8758.392,E2 8758.392} C_VEL
LIN {X 0,Y 363.599,Z 504.426,A -85,B 0,C 180,E1 8754.843,E2 8754.843} C_VEL
LIN {X 0,Y 365.454,Z 505.249,A -85,B 0,C 180,E1 8751.338,E2 8751.338} C_VEL
LIN {X 0,Y 366.569,Z 506.397,A -85,B 0,C 180,E1 8748.61,E2 8748.61} C_VEL
LIN {X 0,Y 367.62,Z 508.256,A -85,B 0,C 180,E1 8745.297,E2 8745.297} C_VEL
LIN {X 0,Y 368.701,Z 509.495,A -85,B 0,C 180,E1 8741.735,E2 8741.735} C_VEL
LIN {X 0,Y 369.368,Z 510.253,A -85,B 0,C 180,E1 8738.248,E2 8738.248} C_VEL
LIN {X 0,Y 369.958,Z 510.669,A -85,B 0,C 180,E1 8734.65,E2 8734.65} C_VEL
LIN {X 0,Y 370.1,Z 510.819,A -85,B 0,C 180,E1 8731.238,E2 8731.238} C_VEL
LIN {X 0,Y 370.126,Z 510.831,A -85,B 0,C 180,E1 8727.833,E2 8727.833} C_VEL
LIN {X 0,Y 369.753,Z 510.578,A -85,B 0,C 180,E1 8724.258,E2 8724.258} C_VEL
LIN {X 0,Y 369.265,Z 510.081,A -85,B 0,C 180,E1 8720.965,E2 8720.965} C_VEL
LIN {X 0,Y 368.376,Z 509.231,A -85,B 0,C 180,E1 8717.3,E2 8717.3} C_VEL
LIN {X 0,Y 367.482,Z 508.007,A -85,B 0,C 180,E1 8714.212,E2 8714.212} C_VEL
LIN {X 0,Y 366.163,Z 505.798,A -85,B 0,C 180,E1 8710.401,E2 8710.401} C_VEL
LIN {X 0,Y 364.783,Z 504.983,A -85,B 0,C 180,E1 8707.435,E2 8707.435} C_VEL
LIN {X 0,Y 362.942,Z 504.027,A -85,B 0,C 180,E1 8703.847,E2 8703.847} C_VEL
LIN {X 0,Y 360.909,Z 502.459,A -85,B 0,C 180,E1 8700.447,E2 8700.447} C_VEL
LIN {X 0,Y 358.974,Z 500.226,A -85,B 0,C 180,E1 8697.263,E2 8697.263} C_VEL
LIN {X 0,Y 357.229,Z 497.862,A -85,B 0,C 180,E1 8694.537,E2 8694.537} C_VEL
LIN {X 0,Y 354.409,Z 496.279,A -85,B 0,C 180,E1 8690.88,E2 8690.88} C_VEL
LIN {X 0,Y 352.034,Z 494.142,A -85,B 0,C 180,E1 8687.842,E2 8687.842} C_VEL
LIN {X 0,Y 349.109,Z 490.457,A -85,B 0,C 180,E1 8684.103,E2 8684.103} C_VEL
LIN {X 0,Y 346.06,Z 488.51,A -85,B 0,C 180,E1 8680.766,E2 8680.766} C_VEL
LIN {X 0,Y 343.321,Z 485.793,A -85,B 0,C 180,E1 8677.704,E2 8677.704} C_VEL
LIN {X 0,Y 341.301,Z 483.188,A -85,B 0,C 180,E1 8675.454,E2 8675.454} C_VEL
LIN {X 0,Y 338.217,Z 481.024,A -85,B 0,C 180,E1 8672.278,E2 8672.278} C_VEL
LIN {X 0,Y 335.186,Z 477.905,A -85,B 0,C 180,E1 8669.191,E2 8669.191} C_VEL
LIN {X 0,Y 333.279,Z 475.838,A -85,B 0,C 180,E1 8667.517,E2 8667.517} C_VEL
LIN {X 0,Y 329.853,Z 473.851,A -85,B 0,C 180,E1 8664.919,E2 8664.919} C_VEL
LIN {X 0,Y 325.352,Z 470.246,A -85,B 0,C 180,E1 8661.83,E2 8661.83} C_VEL
LIN {X 0,Y 322.082,Z 467.27,A -85,B 0,C 180,E1 8659.778,E2 8659.778} C_VEL
LIN {X 0,Y 316.288,Z 462.701,A -85,B 0,C 180,E1 8656.152,E2 8656.152} C_VEL
LIN {X 0,Y 312.628,Z 457.866,A -85,B 0,C 180,E1 8653.125,E2 8653.125} C_VEL
LIN {X 0,Y 309.428,Z 452.491,A -85,B 0,C 180,E1 8649.485,E2 8649.485} C_VEL
LIN {X 0,Y 307.423,Z 448.554,A -85,B 0,C 180,E1 8645.974,E2 8645.974} C_VEL
LIN {X 0,Y 306.085,Z 446.871,A -85,B 0,C 180,E1 8640.561,E2 8640.561} C_VEL
LIN {X 0,Y 306.573,Z 447.733,A -85,B 0,C 180,E1 8636.635,E2 8636.635} C_VEL
LIN {X 0,Y 307.655,Z 449.043,A -85,B 0,C 180,E1 8633.946,E2 8633.946} C_VEL
LIN {X 0,Y 310.094,Z 453.716,A -85,B 0,C 180,E1 8630.067,E2 8630.067} C_VEL
LIN {X 0,Y 312.727,Z 458.585,A -85,B 0,C 180,E1 8627.161,E2 8627.161} C_VEL
LIN {X 0,Y 316.276,Z 465.3,A -85,B 0,C 180,E1 8624.083,E2 8624.083} C_VEL
LIN {X 0,Y 317.65,Z 468.262,A -85,B 0,C 180,E1 8623.024,E2 8623.024} C_VEL
LIN {X 0,Y 305.147,Z 597.769,A -85,B 0,C 180,E1 8620.514,E2 8620.514} C_VEL
LIN {X 0,Y 300.987,Z 622.025,A -85,B 0,C 180,E1 8619.896,E2 8619.896} C_VEL
LIN {X 0,Y 296.267,Z 641.474,A -85,B 0,C 180,E1 8619.246,E2 8619.246} C_VEL
LIN {X 0,Y 289.97,Z 662.329,A -85,B 0,C 180,E1 8618.318,E2 8618.318} C_VEL
LIN {X 0,Y 282.618,Z 681.923,A -85,B 0,C 180,E1 8617.158,E2 8617.158} C_VEL
LIN {X 0,Y 276.82,Z 695.511,A -85,B 0,C 180,E1 8616.172,E2 8616.172} C_VEL
LIN {X 0,Y 273.26,Z 702.404,A -85,B 0,C 180,E1 8615.806,E2 8615.806} C_VEL
LIN {X 0,Y 262.109,Z 719.006,A -85,B 0,C 180,E1 8615.404,E2 8615.404} C_VEL
LIN {X 0,Y 258.166,Z 725.124,A -85,B 0,C 180,E1 8614.924,E2 8614.924} C_VEL
LIN {X 0,Y 247.179,Z 743.159,A -85,B 0,C 180,E1 8612.607,E2 8612.607} C_VEL
LIN {X 0,Y 236.559,Z 758.623,A -85,B 0,C 180,E1 8610.048,E2 8610.048} C_VEL
LIN {X 0,Y 226.801,Z 771.74,A -85,B 0,C 180,E1 8607.352,E2 8607.352} C_VEL
LIN {X 0,Y 214.74,Z 786.745,A -85,B 0,C 180,E1 8603.417,E2 8603.417} C_VEL
LIN {X 0,Y 204.869,Z 798.171,A -85,B 0,C 180,E1 8599.526,E2 8599.526} C_VEL
LIN {X 0,Y 195.875,Z 808.253,A -85,B 0,C 180,E1 8595.196,E2 8595.196} C_VEL
LIN {X 0,Y 185.89,Z 819.21,A -85,B 0,C 180,E1 8588.998,E2 8588.998} C_VEL
LIN {X 0,Y 179.332,Z 826.535,A -85,B 0,C 180,E1 8583.501,E2 8583.501} C_VEL
LIN {X 0,Y 173.861,Z 833.183,A -85,B 0,C 180,E1 8577.02,E2 8577.02} C_VEL
LIN {X 0,Y 170.037,Z 838.577,A -85,B 0,C 180,E1 8569.583,E2 8569.583} C_VEL
LIN {X 0,Y 168.474,Z 841.687,A -85,B 0,C 180,E1 8563.382,E2 8563.382} C_VEL
LIN {X 0,Y 168.024,Z 843.478,A -85,B 0,C 180,E1 8557.866,E2 8557.866} C_VEL
LIN {X 0,Y 168.005,Z 844.319,A -85,B 0,C 180,E1 8552.729,E2 8552.729} C_VEL
LIN {X 0,Y 168.011,Z 844.376,A -85,B 0,C 180,E1 8547.954,E2 8547.954} C_VEL
LIN {X 0,Y 168.009,Z 843.647,A -85,B 0,C 180,E1 8542.821,E2 8542.821} C_VEL
LIN {X 0,Y 168.425,Z 841.827,A -85,B 0,C 180,E1 8536.963,E2 8536.963} C_VEL
LIN {X 0,Y 169.797,Z 838.971,A -85,B 0,C 180,E1 8531.103,E2 8531.103} C_VEL
LIN {X 0,Y 172.94,Z 834.373,A -85,B 0,C 180,E1 8524.411,E2 8524.411} C_VEL
LIN {X 0,Y 178.701,Z 827.28,A -85,B 0,C 180,E1 8517.131,E2 8517.131} C_VEL
LIN {X 0,Y 185.088,Z 820.079,A -85,B 0,C 180,E1 8511.595,E2 8511.595} C_VEL
LIN {X 0,Y 193.915,Z 810.499,A -85,B 0,C 180,E1 8505.888,E2 8505.888} C_VEL
LIN {X 0,Y 203.819,Z 799.37,A -85,B 0,C 180,E1 8500.936,E2 8500.936} C_VEL
LIN {X 0,Y 213.21,Z 788.515,A -85,B 0,C 180,E1 8497.137,E2 8497.137} C_VEL
LIN {X 0,Y 224.789,Z 774.422,A -85,B 0,C 180,E1 8493.259,E2 8493.259} C_VEL
LIN {X 0,Y 235.847,Z 759.618,A -85,B 0,C 180,E1 8490.138,E2 8490.138} C_VEL
LIN {X 0,Y 246.055,Z 744.817,A -85,B 0,C 180,E1 8487.646,E2 8487.646} C_VEL
LIN {X 0,Y 257.488,Z 726.325,A -85,B 0,C 180,E1 8485.211,E2 8485.211} C_VEL
LIN {X 0,Y 266.555,Z 709.738,A -85,B 0,C 180,E1 8483.494,E2 8483.494} C_VEL
LIN {X 0,Y 275.877,Z 690.484,A -85,B 0,C 180,E1 8481.907,E2 8481.907} C_VEL
LIN {X 0,Y 284.141,Z 670.043,A -85,B 0,C 180,E1 8480.61,E2 8480.61} C_VEL
LIN {X 0,Y 290.669,Z 650.974,A -85,B 0,C 180,E1 8479.673,E2 8479.673} C_VEL
LIN {X 0,Y 296.997,Z 627.671,A -85,B 0,C 180,E1 8478.826,E2 8478.826} C_VEL
LIN {X 0,Y 301.027,Z 607.593,A -85,B 0,C 180,E1 8478.286,E2 8478.286} C_VEL
LIN {X 0,Y 304.158,Z 583.536,A -85,B 0,C 180,E1 8477.764,E2 8477.764} C_VEL
LIN {X 0,Y 314.857,Z 473.23,A -85,B 0,C 180,E1 8475.66,E2 8475.66} C_VEL
LIN {X 0,Y 311.377,Z 466.348,A -85,B 0,C 180,E1 8472.541,E2 8472.541} C_VEL
LIN {X 0,Y 309.16,Z 462.178,A -85,B 0,C 180,E1 8470.058,E2 8470.058} C_VEL
LIN {X 0,Y 308.088,Z 460.083,A -85,B 0,C 180,E1 8468.586,E2 8468.586} C_VEL
LIN {X 0,Y 306.301,Z 456.402,A -85,B 0,C 180,E1 8465.244,E2 8465.244} C_VEL
LIN {X 0,Y 305.108,Z 454.807,A -85,B 0,C 180,E1 8460,E2 8460} C_VEL
LIN {X 0,Y 305.692,Z 455.819,A -85,B 0,C 180,E1 8455.874,E2 8455.874} C_VEL
LIN {X 0,Y 306.558,Z 456.904,A -85,B 0,C 180,E1 8453.727,E2 8453.727} C_VEL
LIN {X 0,Y 308.843,Z 461.442,A -85,B 0,C 180,E1 8449.932,E2 8449.932} C_VEL
LIN {X 0,Y 313.262,Z 468.375,A -85,B 0,C 180,E1 8445.395,E2 8445.395} C_VEL
LIN {X 0,Y 318.085,Z 473.356,A -85,B 0,C 180,E1 8441.964,E2 8441.964} C_VEL
LIN {X 0,Y 322.155,Z 476.281,A -85,B 0,C 180,E1 8439.564,E2 8439.564} C_VEL
LIN {X 0,Y 326.456,Z 480.116,A -85,B 0,C 180,E1 8436.728,E2 8436.728} C_VEL
LIN {X 0,Y 330.387,Z 482.786,A -85,B 0,C 180,E1 8433.972,E2 8433.972} C_VEL
LIN {X 0,Y 332.918,Z 484.451,A -85,B 0,C 180,E1 8431.965,E2 8431.965} C_VEL
LIN {X 0,Y 335.83,Z 487.71,A -85,B 0,C 180,E1 8429.197,E2 8429.197} C_VEL
LIN {X 0,Y 339.702,Z 490.807,A -85,B 0,C 180,E1 8425.202,E2 8425.202} C_VEL
LIN {X 0,Y 340.843,Z 491.81,A -85,B 0,C 180,E1 8423.973,E2 8423.973} C_VEL
LIN {X 0,Y 343.857,Z 495.38,A -85,B 0,C 180,E1 8420.662,E2 8420.662} C_VEL
LIN {X 0,Y 346.952,Z 497.816,A -85,B 0,C 180,E1 8417.148,E2 8417.148} C_VEL
LIN {X 0,Y 348.579,Z 498.947,A -85,B 0,C 180,E1 8415.344,E2 8415.344} C_VEL
LIN {X 0,Y 351.171,Z 502.269,A -85,B 0,C 180,E1 8411.996,E2 8411.996} C_VEL
LIN {X 0,Y 353.751,Z 504.453,A -85,B 0,C 180,E1 8408.731,E2 8408.731} C_VEL
LIN {X 0,Y 356.522,Z 506.047,A -85,B 0,C 180,E1 8405.025,E2 8405.025} C_VEL
LIN {X 0,Y 358.591,Z 509.031,A -85,B 0,C 180,E1 8401.742,E2 8401.742} C_VEL
LIN {X 0,Y 360.831,Z 511.196,A -85,B 0,C 180,E1 8398.103,E2 8398.103} C_VEL
LIN {X 0,Y 362.78,Z 512.446,A -85,B 0,C 180,E1 8394.562,E2 8394.562} C_VEL
LIN {X 0,Y 364.693,Z 513.285,A -85,B 0,C 180,E1 8390.788,E2 8390.788} C_VEL
LIN {X 0,Y 365.766,Z 514.827,A -85,B 0,C 180,E1 8387.957,E2 8387.957} C_VEL
LIN {X 0,Y 366.872,Z 516.496,A -85,B 0,C 180,E1 8384.648,E2 8384.648} C_VEL
LIN {X 0,Y 367.841,Z 517.628,A -85,B 0,C 180,E1 8380.968,E2 8380.968} C_VEL
LIN {X 0,Y 368.525,Z 518.273,A -85,B 0,C 180,E1 8377.64,E2 8377.64} C_VEL
LIN {X 0,Y 368.981,Z 518.682,A -85,B 0,C 180,E1 8373.884,E2 8373.884} C_VEL
LIN {X 0,Y 369.146,Z 518.771,A -85,B 0,C 180,E1 8370.776,E2 8370.776} C_VEL
LIN {X 0,Y 369.049,Z 518.691,A -85,B 0,C 180,E1 8366.894,E2 8366.894} C_VEL
LIN {X 0,Y 368.708,Z 518.448,A -85,B 0,C 180,E1 8363.617,E2 8363.617} C_VEL
LIN {X 0,Y 368.022,Z 517.838,A -85,B 0,C 180,E1 8359.829,E2 8359.829} C_VEL
LIN {X 0,Y 367.224,Z 516.929,A -85,B 0,C 180,E1 8356.619,E2 8356.619} C_VEL
LIN {X 0,Y 366.059,Z 515.294,A -85,B 0,C 180,E1 8352.843,E2 8352.843} C_VEL
LIN {X 0,Y 364.92,Z 513.508,A -85,B 0,C 180,E1 8349.805,E2 8349.805} C_VEL
LIN {X 0,Y 363.296,Z 512.698,A -85,B 0,C 180,E1 8346.309,E2 8346.309} C_VEL
LIN {X 0,Y 361.333,Z 511.565,A -85,B 0,C 180,E1 8342.834,E2 8342.834} C_VEL
LIN {X 0,Y 359.34,Z 509.814,A -85,B 0,C 180,E1 8339.391,E2 8339.391} C_VEL
LIN {X 0,Y 357.078,Z 506.936,A -85,B 0,C 180,E1 8335.856,E2 8335.856} C_VEL
LIN {X 0,Y 356.057,Z 505.71,A -85,B 0,C 180,E1 8334.248,E2 8334.248} C_VEL
LIN {X 0,Y 353.245,Z 504.113,A -85,B 0,C 180,E1 8330.653,E2 8330.653} C_VEL
LIN {X 0,Y 350.802,Z 501.859,A -85,B 0,C 180,E1 8327.509,E2 8327.509} C_VEL
LIN {X 0,Y 348.061,Z 498.379,A -85,B 0,C 180,E1 8324.042,E2 8324.042} C_VEL
LIN {X 0,Y 345.008,Z 496.44,A -85,B 0,C 180,E1 8320.697,E2 8320.697} C_VEL
LIN {X 0,Y 342.107,Z 493.546,A -85,B 0,C 180,E1 8317.438,E2 8317.438} C_VEL
LIN {X 0,Y 340.049,Z 491.004,A -85,B 0,C 180,E1 8315.176,E2 8315.176} C_VEL
LIN {X 0,Y 336.536,Z 488.377,A -85,B 0,C 180,E1 8311.527,E2 8311.527} C_VEL
LIN {X 0,Y 333.403,Z 485.064,A -85,B 0,C 180,E1 8308.479,E2 8308.479} C_VEL
LIN {X 0,Y 331.914,Z 483.626,A -85,B 0,C 180,E1 8307.251,E2 8307.251} C_VEL
LIN {X 0,Y 328.256,Z 481.429,A -85,B 0,C 180,E1 8304.472,E2 8304.472} C_VEL
LIN {X 0,Y 323.716,Z 477.829,A -85,B 0,C 180,E1 8301.47,E2 8301.47} C_VEL
LIN {X 0,Y 320.558,Z 474.986,A -85,B 0,C 180,E1 8299.496,E2 8299.496} C_VEL
LIN {X 0,Y 314.718,Z 470.255,A -85,B 0,C 180,E1 8295.761,E2 8295.761} C_VEL
LIN {X 0,Y 311.266,Z 465.557,A -85,B 0,C 180,E1 8292.806,E2 8292.806} C_VEL
LIN {X 0,Y 308.178,Z 460.199,A -85,B 0,C 180,E1 8289.147,E2 8289.147} C_VEL
LIN {X 0,Y 306.36,Z 456.447,A -85,B 0,C 180,E1 8285.807,E2 8285.807} C_VEL
LIN {X 0,Y 305.11,Z 454.811,A -85,B 0,C 180,E1 8280.563,E2 8280.563} C_VEL
LIN {X 0,Y 305.597,Z 455.698,A -85,B 0,C 180,E1 8276.624,E2 8276.624} C_VEL
LIN {X 0,Y 306.544,Z 456.867,A -85,B 0,C 180,E1 8274.197,E2 8274.197} C_VEL
LIN {X 0,Y 308.816,Z 461.415,A -85,B 0,C 180,E1 8270.402,E2 8270.402} C_VEL
LIN {X 0,Y 311.377,Z 466.348,A -85,B 0,C 180,E1 8267.459,E2 8267.459} C_VEL
LIN {X 0,Y 314.875,Z 473.272,A -85,B 0,C 180,E1 8264.325,E2 8264.325} C_VEL
LIN {X 0,Y 302.55,Z 597.633,A -85,B 0,C 180,E1 8261.946,E2 8261.946} C_VEL
LIN {X 0,Y 298.315,Z 621.811,A -85,B 0,C 180,E1 8261.345,E2 8261.345} C_VEL
LIN {X 0,Y 293.437,Z 641.515,A -85,B 0,C 180,E1 8260.704,E2 8260.704} C_VEL
LIN {X 0,Y 286.897,Z 662.622,A -85,B 0,C 180,E1 8259.787,E2 8259.787} C_VEL
LIN {X 0,Y 279.162,Z 682.661,A -85,B 0,C 180,E1 8258.623,E2 8258.623} C_VEL
LIN {X 0,Y 271.278,Z 700.321,A -85,B 0,C 180,E1 8257.327,E2 8257.327} C_VEL
LIN {X 0,Y 261.01,Z 720.138,A -85,B 0,C 180,E1 8255.474,E2 8255.474} C_VEL
LIN {X 0,Y 258.166,Z 725.124,A -85,B 0,C 180,E1 8254.924,E2 8254.924} C_VEL
LIN {X 0,Y 254.083,Z 731.364,A -85,B 0,C 180,E1 8254.394,E2 8254.394} C_VEL
LIN {X 0,Y 242.133,Z 745.765,A -85,B 0,C 180,E1 8253.619,E2 8253.619} C_VEL
LIN {X 0,Y 237.636,Z 751.459,A -85,B 0,C 180,E1 8253,E2 8253} C_VEL
LIN {X 0,Y 237.078,Z 752.262,A -85,B 0,C 180,E1 8252.877,E2 8252.877} C_VEL
LIN {X 0,Y 225.1,Z 768.158,A -85,B 0,C 180,E1 8249.872,E2 8249.872} C_VEL
LIN {X 0,Y 214.89,Z 780.655,A -85,B 0,C 180,E1 8246.877,E2 8246.877} C_VEL
LIN {X 0,Y 203.088,Z 794.217,A -85,B 0,C 180,E1 8242.731,E2 8242.731} C_VEL
LIN {X 0,Y 192.266,Z 805.725,A -85,B 0,C 180,E1 8238.042,E2 8238.042} C_VEL
LIN {X 0,Y 183.6,Z 814.739,A -85,B 0,C 180,E1 8233.327,E2 8233.327} C_VEL
LIN {X 0,Y 174.659,Z 824.045,A -85,B 0,C 180,E1 8226.947,E2 8226.947} C_VEL
LIN {X 0,Y 168.21,Z 830.957,A -85,B 0,C 180,E1 8220.47,E2 8220.47} C_VEL
LIN {X 0,Y 163.954,Z 836.074,A -85,B 0,C 180,E1 8214.116,E2 8214.116} C_VEL
LIN {X 0,Y 161.003,Z 840.588,A -85,B 0,C 180,E1 8206.227,E2 8206.227} C_VEL
LIN {X 0,Y 160.072,Z 842.988,A -85,B 0,C 180,E1 8199.279,E2 8199.279} C_VEL
LIN {X 0,Y 159.999,Z 844.013,A -85,B 0,C 180,E1 8193.583,E2 8193.583} C_VEL
LIN {X 0,Y 160.02,Z 844.183,A -85,B 0,C 180,E1 8188.568,E2 8188.568} C_VEL
LIN {X 0,Y 160.01,Z 843.481,A -85,B 0,C 180,E1 8182.821,E2 8182.821} C_VEL
LIN {X 0,Y 160.457,Z 841.715,A -85,B 0,C 180,E1 8176.67,E2 8176.67} C_VEL
LIN {X 0,Y 162.066,Z 838.717,A -85,B 0,C 180,E1 8170.165,E2 8170.165} C_VEL
LIN {X 0,Y 165.603,Z 834.042,A -85,B 0,C 180,E1 8163.076,E2 8163.076} C_VEL
LIN {X 0,Y 171.802,Z 827.022,A -85,B 0,C 180,E1 8155.632,E2 8155.632} C_VEL
LIN {X 0,Y 178.662,Z 819.822,A -85,B 0,C 180,E1 8149.942,E2 8149.942} C_VEL
LIN {X 0,Y 188.047,Z 810.242,A -85,B 0,C 180,E1 8144.128,E2 8144.128} C_VEL
LIN {X 0,Y 198.489,Z 799.116,A -85,B 0,C 180,E1 8139.129,E2 8139.129} C_VEL
LIN {X 0,Y 208.324,Z 788.262,A -85,B 0,C 180,E1 8135.324,E2 8135.324} C_VEL
LIN {X 0,Y 220.487,Z 774.021,A -85,B 0,C 180,E1 8131.433,E2 8131.433} C_VEL
LIN {X 0,Y 231.828,Z 759.366,A -85,B 0,C 180,E1 8128.38,E2 8128.38} C_VEL
LIN {X 0,Y 242.362,Z 744.567,A -85,B 0,C 180,E1 8125.93,E2 8125.93} C_VEL
LIN {X 0,Y 254.34,Z 725.696,A -85,B 0,C 180,E1 8123.505,E2 8123.505} C_VEL
LIN {X 0,Y 263.46,Z 709.414,A -85,B 0,C 180,E1 8121.864,E2 8121.864} C_VEL
LIN {X 0,Y 272.956,Z 690.23,A -85,B 0,C 180,E1 8120.328,E2 8120.328} C_VEL
LIN {X 0,Y 281.399,Z 669.798,A -85,B 0,C 180,E1 8119.07,E2 8119.07} C_VEL
LIN {X 0,Y 288.273,Z 650.073,A -85,B 0,C 180,E1 8118.135,E2 8118.135} C_VEL
LIN {X 0,Y 294.583,Z 627.073,A -85,B 0,C 180,E1 8117.336,E2 8117.336} C_VEL
LIN {X 0,Y 298.712,Z 606.749,A -85,B 0,C 180,E1 8116.807,E2 8116.807} C_VEL
LIN {X 0,Y 301.991,Z 581.387,A -85,B 0,C 180,E1 8116.276,E2 8116.276} C_VEL
LIN {X 0,Y 312.198,Z 478.507,A -85,B 0,C 180,E1 8114.324,E2 8114.324} C_VEL
LIN {X 0,Y 309.09,Z 472.106,A -85,B 0,C 180,E1 8111.192,E2 8111.192} C_VEL
LIN {X 0,Y 306.852,Z 467.787,A -85,B 0,C 180,E1 8108.243,E2 8108.243} C_VEL
LIN {X 0,Y 305.242,Z 464.294,A -85,B 0,C 180,E1 8105.074,E2 8105.074} C_VEL
LIN {X 0,Y 304.133,Z 462.747,A -85,B 0,C 180,E1 8100,E2 8100} C_VEL
LIN {X 0,Y 304.659,Z 463.706,A -85,B 0,C 180,E1 8096.048,E2 8096.048} C_VEL
LIN {X 0,Y 305.449,Z 464.716,A -85,B 0,C 180,E1 8093.987,E2 8093.987} C_VEL
LIN {X 0,Y 307.575,Z 469.142,A -85,B 0,C 180,E1 8090.268,E2 8090.268} C_VEL
LIN {X 0,Y 311.753,Z 475.92,A -85,B 0,C 180,E1 8085.797,E2 8085.797} C_VEL
LIN {X 0,Y 316.579,Z 481.053,A -85,B 0,C 180,E1 8082.255,E2 8082.255} C_VEL
LIN {X 0,Y 320.772,Z 484.116,A -85,B 0,C 180,E1 8079.758,E2 8079.758} C_VEL
LIN {X 0,Y 325.271,Z 488.036,A -85,B 0,C 180,E1 8076.83,E2 8076.83} C_VEL
LIN {X 0,Y 328.957,Z 490.548,A -85,B 0,C 180,E1 8074.237,E2 8074.237} C_VEL
LIN {X 0,Y 331.535,Z 492.181,A -85,B 0,C 180,E1 8072.228,E2 8072.228} C_VEL
LIN {X 0,Y 334.615,Z 495.546,A -85,B 0,C 180,E1 8069.378,E2 8069.378} C_VEL
LIN {X 0,Y 338.323,Z 498.527,A -85,B 0,C 180,E1 8065.635,E2 8065.635} C_VEL
LIN {X 0,Y 339.596,Z 499.556,A -85,B 0,C 180,E1 8064.237,E2 8064.237} C_VEL
LIN {X 0,Y 342.281,Z 502.859,A -85,B 0,C 180,E1 8061.254,E2 8061.254} C_VEL
LIN {X 0,Y 345.744,Z 505.637,A -85,B 0,C 180,E1 8057.413,E2 8057.413} C_VEL
LIN {X 0,Y 347.535,Z 506.931,A -85,B 0,C 180,E1 8055.414,E2 8055.414} C_VEL
LIN {X 0,Y 350.135,Z 510.212,A -85,B 0,C 180,E1 8052.058,E2 8052.058} C_VEL
LIN {X 0,Y 352.724,Z 512.383,A -85,B 0,C 180,E1 8048.782,E2 8048.782} C_VEL
LIN {X 0,Y 355.542,Z 514.099,A -85,B 0,C 180,E1 8045.007,E2 8045.007} C_VEL
LIN {X 0,Y 357.63,Z 517.041,A -85,B 0,C 180,E1 8041.708,E2 8041.708} C_VEL
LIN {X 0,Y 359.931,Z 519.212,A -85,B 0,C 180,E1 8037.948,E2 8037.948} C_VEL
LIN {X 0,Y 361.847,Z 520.413,A -85,B 0,C 180,E1 8034.486,E2 8034.486} C_VEL
LIN {X 0,Y 363.785,Z 521.311,A -85,B 0,C 180,E1 8030.597,E2 8030.597} C_VEL
LIN {X 0,Y 364.868,Z 522.951,A -85,B 0,C 180,E1 8027.708,E2 8027.708} C_VEL
LIN {X 0,Y 366.09,Z 524.614,A -85,B 0,C 180,E1 8024.172,E2 8024.172} C_VEL
LIN {X 0,Y 366.923,Z 525.657,A -85,B 0,C 180,E1 8020.678,E2 8020.678} C_VEL
LIN {X 0,Y 367.677,Z 526.267,A -85,B 0,C 180,E1 8017.186,E2 8017.186} C_VEL
LIN {X 0,Y 368.025,Z 526.626,A -85,B 0,C 180,E1 8013.582,E2 8013.582} C_VEL
LIN {X 0,Y 368.235,Z 526.746,A -85,B 0,C 180,E1 8010.156,E2 8010.156} C_VEL
LIN {X 0,Y 368.038,Z 526.627,A -85,B 0,C 180,E1 8006.574,E2 8006.574} C_VEL
LIN {X 0,Y 367.708,Z 526.308,A -85,B 0,C 180,E1 8003.129,E2 8003.129} C_VEL
LIN {X 0,Y 366.985,Z 525.727,A -85,B 0,C 180,E1 7999.593,E2 7999.593} C_VEL
LIN {X 0,Y 366.173,Z 524.747,A -85,B 0,C 180,E1 7996.258,E2 7996.258} C_VEL
LIN {X 0,Y 364.992,Z 523.14,A -85,B 0,C 180,E1 7992.627,E2 7992.627} C_VEL
LIN {X 0,Y 363.919,Z 521.437,A -85,B 0,C 180,E1 7989.747,E2 7989.747} C_VEL
LIN {X 0,Y 362.272,Z 520.621,A -85,B 0,C 180,E1 7986.238,E2 7986.238} C_VEL
LIN {X 0,Y 360.307,Z 519.483,A -85,B 0,C 180,E1 7982.751,E2 7982.751} C_VEL
LIN {X 0,Y 358.277,Z 517.705,A -85,B 0,C 180,E1 7979.266,E2 7979.266} C_VEL
LIN {X 0,Y 356.074,Z 514.93,A -85,B 0,C 180,E1 7975.835,E2 7975.835} C_VEL
LIN {X 0,Y 354.979,Z 513.618,A -85,B 0,C 180,E1 7974.137,E2 7974.137} C_VEL
LIN {X 0,Y 352.184,Z 512.018,A -85,B 0,C 180,E1 7970.553,E2 7970.553} C_VEL
LIN {X 0,Y 349.666,Z 509.679,A -85,B 0,C 180,E1 7967.297,E2 7967.297} C_VEL
LIN {X 0,Y 346.819,Z 506.213,A -85,B 0,C 180,E1 7963.781,E2 7963.781} C_VEL
LIN {X 0,Y 343.957,Z 504.369,A -85,B 0,C 180,E1 7960.628,E2 7960.628} C_VEL
LIN {X 0,Y 340.975,Z 501.403,A -85,B 0,C 180,E1 7957.267,E2 7957.267} C_VEL
LIN {X 0,Y 339.002,Z 498.926,A -85,B 0,C 180,E1 7955.109,E2 7955.109} C_VEL
LIN {X 0,Y 335.452,Z 496.303,A -85,B 0,C 180,E1 7951.44,E2 7951.44} C_VEL
LIN {X 0,Y 332.295,Z 493.036,A -85,B 0,C 180,E1 7948.386,E2 7948.386} C_VEL
LIN {X 0,Y 330.573,Z 491.415,A -85,B 0,C 180,E1 7946.981,E2 7946.981} C_VEL
LIN {X 0,Y 326.295,Z 488.803,A -85,B 0,C 180,E1 7943.859,E2 7943.859} C_VEL
LIN {X 0,Y 322.1,Z 485.412,A -85,B 0,C 180,E1 7941.105,E2 7941.105} C_VEL
LIN {X 0,Y 318.747,Z 482.522,A -85,B 0,C 180,E1 7939.04,E2 7939.04} C_VEL
LIN {X 0,Y 313.049,Z 477.671,A -85,B 0,C 180,E1 7935.278,E2 7935.278} C_VEL
LIN {X 0,Y 309.823,Z 473.13,A -85,B 0,C 180,E1 7932.393,E2 7932.393} C_VEL
LIN {X 0,Y 306.939,Z 467.906,A -85,B 0,C 180,E1 7928.807,E2 7928.807} C_VEL
LIN {X 0,Y 305.215,Z 464.276,A -85,B 0,C 180,E1 7925.451,E2 7925.451} C_VEL
LIN {X 0,Y 304.131,Z 462.754,A -85,B 0,C 180,E1 7920.377,E2 7920.377} C_VEL
LIN {X 0,Y 304.676,Z 463.741,A -85,B 0,C 180,E1 7916.425,E2 7916.425} C_VEL
LIN {X 0,Y 305.471,Z 464.798,A -85,B 0,C 180,E1 7914.365,E2 7914.365} C_VEL
LIN {X 0,Y 307.612,Z 469.268,A -85,B 0,C 180,E1 7910.647,E2 7910.647} C_VEL
LIN {X 0,Y 309.994,Z 474.025,A -85,B 0,C 180,E1 7907.804,E2 7907.804} C_VEL
LIN {X 0,Y 312.227,Z 478.745,A -85,B 0,C 180,E1 7905.634,E2 7905.634} C_VEL
LIN {X 0,Y 300.144,Z 597.497,A -85,B 0,C 180,E1 7903.402,E2 7903.402} C_VEL
LIN {X 0,Y 295.842,Z 621.578,A -85,B 0,C 180,E1 7902.818,E2 7902.818} C_VEL
LIN {X 0,Y 290.878,Z 641.275,A -85,B 0,C 180,E1 7902.2,E2 7902.2} C_VEL
LIN {X 0,Y 284.437,Z 661.726,A -85,B 0,C 180,E1 7901.344,E2 7901.344} C_VEL
LIN {X 0,Y 276.621,Z 681.7,A -85,B 0,C 180,E1 7900.23,E2 7900.23} C_VEL
LIN {X 0,Y 268.788,Z 698.956,A -85,B 0,C 180,E1 7899.013,E2 7899.013} C_VEL
LIN {X 0,Y 258.951,Z 717.826,A -85,B 0,C 180,E1 7897.338,E2 7897.338} C_VEL
LIN {X 0,Y 248.582,Z 735.044,A -85,B 0,C 180,E1 7895.368,E2 7895.368} C_VEL
LIN {X 0,Y 238.552,Z 750.097,A -85,B 0,C 180,E1 7893.219,E2 7893.219} C_VEL
LIN {X 0,Y 237.078,Z 752.262,A -85,B 0,C 180,E1 7892.877,E2 7892.877} C_VEL
LIN {X 0,Y 232.626,Z 757.886,A -85,B 0,C 180,E1 7892.147,E2 7892.147} C_VEL
LIN {X 0,Y 218.835,Z 771.471,A -85,B 0,C 180,E1 7890.747,E2 7890.747} C_VEL
LIN {X 0,Y 214.036,Z 776.386,A -85,B 0,C 180,E1 7889.793,E2 7889.793} C_VEL
LIN {X 0,Y 202.989,Z 788.727,A -85,B 0,C 180,E1 7886.348,E2 7886.348} C_VEL
LIN {X 0,Y 192.147,Z 800.143,A -85,B 0,C 180,E1 7882.272,E2 7882.272} C_VEL
LIN {X 0,Y 180.23,Z 811.985,A -85,B 0,C 180,E1 7876.613,E2 7876.613} C_VEL
LIN {X 0,Y 171.565,Z 820.369,A -85,B 0,C 180,E1 7871.254,E2 7871.254} C_VEL
LIN {X 0,Y 163.282,Z 828.608,A -85,B 0,C 180,E1 7864.288,E2 7864.288} C_VEL
LIN {X 0,Y 157.342,Z 834.802,A -85,B 0,C 180,E1 7856.819,E2 7856.819} C_VEL
LIN {X 0,Y 154.099,Z 838.856,A -85,B 0,C 180,E1 7850.113,E2 7850.113} C_VEL
LIN {X 0,Y 152.338,Z 842.025,A -85,B 0,C 180,E1 7842.509,E2 7842.509} C_VEL
LIN {X 0,Y 151.994,Z 843.647,A -85,B 0,C 180,E1 7835.284,E2 7835.284} C_VEL
LIN {X 0,Y 152.03,Z 843.99,A -85,B 0,C 180,E1 7829.246,E2 7829.246} C_VEL
LIN {X 0,Y 152.012,Z 843.315,A -85,B 0,C 180,E1 7822.821,E2 7822.821} C_VEL
LIN {X 0,Y 152.558,Z 841.448,A -85,B 0,C 180,E1 7815.925,E2 7815.925} C_VEL
LIN {X 0,Y 154.378,Z 838.462,A -85,B 0,C 180,E1 7809.133,E2 7809.133} C_VEL
LIN {X 0,Y 158.292,Z 833.786,A -85,B 0,C 180,E1 7801.723,E2 7801.723} C_VEL
LIN {X 0,Y 165.03,Z 826.765,A -85,B 0,C 180,E1 7794.008,E2 7794.008} C_VEL
LIN {X 0,Y 172.395,Z 819.565,A -85,B 0,C 180,E1 7788.167,E2 7788.167} C_VEL
LIN {X 0,Y 182.367,Z 809.985,A -85,B 0,C 180,E1 7782.257,E2 7782.257} C_VEL
LIN {X 0,Y 193.369,Z 798.862,A -85,B 0,C 180,E1 7777.225,E2 7777.225} C_VEL
LIN {X 0,Y 203.658,Z 788.008,A -85,B 0,C 180,E1 7773.427,E2 7773.427} C_VEL
LIN {X 0,Y 216.184,Z 773.91,A -85,B 0,C 180,E1 7769.602,E2 7769.602} C_VEL
LIN {X 0,Y 228.035,Z 759.115,A -85,B 0,C 180,E1 7766.562,E2 7766.562} C_VEL
LIN {X 0,Y 239.291,Z 743.764,A -85,B 0,C 180,E1 7764.082,E2 7764.082} C_VEL
LIN {X 0,Y 251.382,Z 725.138,A -85,B 0,C 180,E1 7761.766,E2 7761.766} C_VEL
LIN {X 0,Y 260.919,Z 708.474,A -85,B 0,C 180,E1 7760.144,E2 7760.144} C_VEL
LIN {X 0,Y 270.676,Z 689.063,A -85,B 0,C 180,E1 7758.654,E2 7758.654} C_VEL
LIN {X 0,Y 278.864,Z 669.553,A -85,B 0,C 180,E1 7757.502,E2 7757.502} C_VEL
LIN {X 0,Y 285.868,Z 649.831,A -85,B 0,C 180,E1 7756.6,E2 7756.6} C_VEL
LIN {X 0,Y 292.289,Z 626.834,A -85,B 0,C 180,E1 7755.832,E2 7755.832} C_VEL
LIN {X 0,Y 296.516,Z 606.362,A -85,B 0,C 180,E1 7755.317,E2 7755.317} C_VEL
LIN {X 0,Y 299.889,Z 580.628,A -85,B 0,C 180,E1 7754.792,E2 7754.792} C_VEL
LIN {X 0,Y 309.731,Z 484.096,A -85,B 0,C 180,E1 7753.012,E2 7753.012} C_VEL
LIN {X 0,Y 307.308,Z 478.993,A -85,B 0,C 180,E1 7750.308,E2 7750.308} C_VEL
LIN {X 0,Y 305.627,Z 475.49,A -85,B 0,C 180,E1 7747.898,E2 7747.898} C_VEL
LIN {X 0,Y 304.186,Z 472.187,A -85,B 0,C 180,E1 7744.903,E2 7744.903} C_VEL
LIN {X 0,Y 303.155,Z 470.691,A -85,B 0,C 180,E1 7739.811,E2 7739.811} C_VEL
LIN {X 0,Y 303.867,Z 471.898,A -85,B 0,C 180,E1 7735.471,E2 7735.471} C_VEL
LIN {X 0,Y 304.381,Z 472.648,A -85,B 0,C 180,E1 7734.155,E2 7734.155} C_VEL
LIN {X 0,Y 306.38,Z 476.995,A -85,B 0,C 180,E1 7730.514,E2 7730.514} C_VEL
LIN {X 0,Y 310.458,Z 483.77,A -85,B 0,C 180,E1 7726.022,E2 7726.022} C_VEL
LIN {X 0,Y 315.354,Z 488.959,A -85,B 0,C 180,E1 7722.375,E2 7722.375} C_VEL
LIN {X 0,Y 319.381,Z 491.949,A -85,B 0,C 180,E1 7719.952,E2 7719.952} C_VEL
LIN {X 0,Y 324.088,Z 495.956,A -85,B 0,C 180,E1 7716.933,E2 7716.933} C_VEL
LIN {X 0,Y 327.797,Z 498.448,A -85,B 0,C 180,E1 7714.334,E2 7714.334} C_VEL
LIN {X 0,Y 330.289,Z 500.039,A -85,B 0,C 180,E1 7712.409,E2 7712.409} C_VEL
LIN {X 0,Y 333.257,Z 503.217,A -85,B 0,C 180,E1 7709.732,E2 7709.732} C_VEL
LIN {X 0,Y 336.678,Z 506.1,A -85,B 0,C 180,E1 7706.255,E2 7706.255} C_VEL
LIN {X 0,Y 338.44,Z 507.425,A -85,B 0,C 180,E1 7704.409,E2 7704.409} C_VEL
LIN {X 0,Y 341.171,Z 510.754,A -85,B 0,C 180,E1 7701.374,E2 7701.374} C_VEL
LIN {X 0,Y 344.732,Z 513.576,A -85,B 0,C 180,E1 7697.449,E2 7697.449} C_VEL
LIN {X 0,Y 346.399,Z 514.798,A -85,B 0,C 180,E1 7695.576,E2 7695.576} C_VEL
LIN {X 0,Y 349.135,Z 518.192,A -85,B 0,C 180,E1 7692.076,E2 7692.076} C_VEL
LIN {X 0,Y 351.811,Z 520.386,A -85,B 0,C 180,E1 7688.699,E2 7688.699} C_VEL
LIN {X 0,Y 354.488,Z 522.015,A -85,B 0,C 180,E1 7685.119,E2 7685.119} C_VEL
LIN {X 0,Y 356.577,Z 524.947,A -85,B 0,C 180,E1 7681.813,E2 7681.813} C_VEL
LIN {X 0,Y 358.886,Z 527.107,A -85,B 0,C 180,E1 7678.088,E2 7678.088} C_VEL
LIN {X 0,Y 360.828,Z 528.336,A -85,B 0,C 180,E1 7674.56,E2 7674.56} C_VEL
LIN {X 0,Y 362.726,Z 529.173,A -85,B 0,C 180,E1 7670.829,E2 7670.829} C_VEL
LIN {X 0,Y 363.816,Z 530.791,A -85,B 0,C 180,E1 7667.926,E2 7667.926} C_VEL
LIN {X 0,Y 364.936,Z 532.415,A -85,B 0,C 180,E1 7664.599,E2 7664.599} C_VEL
LIN {X 0,Y 365.91,Z 533.551,A -85,B 0,C 180,E1 7660.868,E2 7660.868} C_VEL
LIN {X 0,Y 366.607,Z 534.163,A -85,B 0,C 180,E1 7657.522,E2 7657.522} C_VEL
LIN {X 0,Y 367.031,Z 534.562,A -85,B 0,C 180,E1 7653.905,E2 7653.905} C_VEL
LIN {X 0,Y 367.196,Z 534.652,A -85,B 0,C 180,E1 7650.78,E2 7650.78} C_VEL
LIN {X 0,Y 367.098,Z 534.572,A -85,B 0,C 180,E1 7646.877,E2 7646.877} C_VEL
LIN {X 0,Y 366.756,Z 534.327,A -85,B 0,C 180,E1 7643.583,E2 7643.583} C_VEL
LIN {X 0,Y 366.056,Z 533.712,A -85,B 0,C 180,E1 7639.774,E2 7639.774} C_VEL
LIN {X 0,Y 365.255,Z 532.806,A -85,B 0,C 180,E1 7636.545,E2 7636.545} C_VEL
LIN {X 0,Y 364.06,Z 531.165,A -85,B 0,C 180,E1 7632.746,E2 7632.746} C_VEL
LIN {X 0,Y 362.918,Z 529.365,A -85,B 0,C 180,E1 7629.688,E2 7629.688} C_VEL
LIN {X 0,Y 361.144,Z 528.494,A -85,B 0,C 180,E1 7625.985,E2 7625.985} C_VEL
LIN {X 0,Y 359.246,Z 527.375,A -85,B 0,C 180,E1 7622.603,E2 7622.603} C_VEL
LIN {X 0,Y 357.106,Z 525.482,A -85,B 0,C 180,E1 7618.955,E2 7618.955} C_VEL
LIN {X 0,Y 354.867,Z 522.633,A -85,B 0,C 180,E1 7615.507,E2 7615.507} C_VEL
LIN {X 0,Y 353.886,Z 521.519,A -85,B 0,C 180,E1 7614.009,E2 7614.009} C_VEL
LIN {X 0,Y 351.235,Z 520.003,A -85,B 0,C 180,E1 7610.595,E2 7610.595} C_VEL
LIN {X 0,Y 348.582,Z 517.572,A -85,B 0,C 180,E1 7607.173,E2 7607.173} C_VEL
LIN {X 0,Y 345.759,Z 514.128,A -85,B 0,C 180,E1 7603.704,E2 7603.704} C_VEL
LIN {X 0,Y 342.787,Z 512.198,A -85,B 0,C 180,E1 7600.423,E2 7600.423} C_VEL
LIN {X 0,Y 339.673,Z 509.049,A -85,B 0,C 180,E1 7596.905,E2 7596.905} C_VEL
LIN {X 0,Y 337.772,Z 506.746,A -85,B 0,C 180,E1 7594.841,E2 7594.841} C_VEL
LIN {X 0,Y 334.011,Z 503.903,A -85,B 0,C 180,E1 7590.989,E2 7590.989} C_VEL
LIN {X 0,Y 330.868,Z 500.699,A -85,B 0,C 180,E1 7588.07,E2 7588.07} C_VEL
LIN {X 0,Y 329.239,Z 499.203,A -85,B 0,C 180,E1 7586.709,E2 7586.709} C_VEL
LIN {X 0,Y 325.103,Z 496.713,A -85,B 0,C 180,E1 7583.759,E2 7583.759} C_VEL
LIN {X 0,Y 320.888,Z 493.356,A -85,B 0,C 180,E1 7580.998,E2 7580.998} C_VEL
LIN {X 0,Y 317.211,Z 490.23,A -85,B 0,C 180,E1 7578.754,E2 7578.754} C_VEL
LIN {X 0,Y 311.623,Z 485.361,A -85,B 0,C 180,E1 7574.968,E2 7574.968} C_VEL
LIN {X 0,Y 308.396,Z 480.7,A -85,B 0,C 180,E1 7571.976,E2 7571.976} C_VEL
LIN {X 0,Y 305.711,Z 475.613,A -85,B 0,C 180,E1 7568.463,E2 7568.463} C_VEL
LIN {X 0,Y 304.16,Z 472.169,A -85,B 0,C 180,E1 7565.281,E2 7565.281} C_VEL
LIN {X 0,Y 303.156,Z 470.694,A -85,B 0,C 180,E1 7560.378,E2 7560.378} C_VEL
LIN {X 0,Y 303.7,Z 471.704,A -85,B 0,C 180,E1 7556.414,E2 7556.414} C_VEL
LIN {X 0,Y 304.368,Z 472.607,A -85,B 0,C 180,E1 7554.628,E2 7554.628} C_VEL
LIN {X 0,Y 306.353,Z 476.965,A -85,B 0,C 180,E1 7550.987,E2 7550.987} C_VEL
LIN {X 0,Y 308.643,Z 481.742,A -85,B 0,C 180,E1 7548.129,E2 7548.129} C_VEL
LIN {X 0,Y 309.729,Z 484.316,A -85,B 0,C 180,E1 7546.967,E2 7546.967} C_VEL
LIN {X 0,Y 297.936,Z 597.361,A -85,B 0,C 180,E1 7544.881,E2 7544.881} C_VEL
LIN {X 0,Y 293.541,Z 621.458,A -85,B 0,C 180,E1 7544.313,E2 7544.313} C_VEL
LIN {X 0,Y 288.521,Z 641.036,A -85,B 0,C 180,E1 7543.721,E2 7543.721} C_VEL
LIN {X 0,Y 281.489,Z 662.762,A -85,B 0,C 180,E1 7542.837,E2 7542.837} C_VEL
LIN {X 0,Y 273.679,Z 682.164,A -85,B 0,C 180,E1 7541.779,E2 7541.779} C_VEL
LIN {X 0,Y 265.144,Z 700.446,A -85,B 0,C 180,E1 7540.514,E2 7540.514} C_VEL
LIN {X 0,Y 254.265,Z 720.326,A -85,B 0,C 180,E1 7538.739,E2 7538.739} C_VEL
LIN {X 0,Y 244.483,Z 736.024,A -85,B 0,C 180,E1 7536.948,E2 7536.948} C_VEL
LIN {X 0,Y 233.188,Z 752.381,A -85,B 0,C 180,E1 7534.61,E2 7534.61} C_VEL
LIN {X 0,Y 221.289,Z 767.658,A -85,B 0,C 180,E1 7531.77,E2 7531.77} C_VEL
LIN {X 0,Y 214.036,Z 776.386,A -85,B 0,C 180,E1 7529.793,E2 7529.793} C_VEL
LIN {X 0,Y 209.214,Z 781.246,A -85,B 0,C 180,E1 7528.769,E2 7528.769} C_VEL
LIN {X 0,Y 194.754,Z 793.05,A -85,B 0,C 180,E1 7526.621,E2 7526.621} C_VEL
LIN {X 0,Y 189.925,Z 797.18,A -85,B 0,C 180,E1 7525.331,E2 7525.331} C_VEL
LIN {X 0,Y 179.213,Z 807.487,A -85,B 0,C 180,E1 7520.849,E2 7520.849} C_VEL
LIN {X 0,Y 167.285,Z 818.44,A -85,B 0,C 180,E1 7514.37,E2 7514.37} C_VEL
LIN {X 0,Y 159.197,Z 825.766,A -85,B 0,C 180,E1 7508.445,E2 7508.445} C_VEL
LIN {X 0,Y 152.215,Z 832.414,A -85,B 0,C 180,E1 7501.26,E2 7501.26} C_VEL
LIN {X 0,Y 147.073,Z 837.813,A -85,B 0,C 180,E1 7492.799,E2 7492.799} C_VEL
LIN {X 0,Y 144.82,Z 840.928,A -85,B 0,C 180,E1 7485.62,E2 7485.62} C_VEL
LIN {X 0,Y 144.055,Z 842.811,A -85,B 0,C 180,E1 7478.783,E2 7478.783} C_VEL
LIN {X 0,Y 144.013,Z 843.602,A -85,B 0,C 180,E1 7472.786,E2 7472.786} C_VEL
LIN {X 0,Y 144.017,Z 843.63,A -85,B 0,C 180,E1 7467.613,E2 7467.613} C_VEL
LIN {X 0,Y 144.042,Z 842.896,A -85,B 0,C 180,E1 7461.618,E2 7461.618} C_VEL
LIN {X 0,Y 144.743,Z 841.069,A -85,B 0,C 180,E1 7454.782,E2 7454.782} C_VEL
LIN {X 0,Y 146.903,Z 838.01,A -85,B 0,C 180,E1 7447.596,E2 7447.596} C_VEL
LIN {X 0,Y 151.924,Z 832.726,A -85,B 0,C 180,E1 7439.114,E2 7439.114} C_VEL
LIN {X 0,Y 158.796,Z 826.138,A -85,B 0,C 180,E1 7431.9,E2 7431.9} C_VEL
LIN {X 0,Y 166.792,Z 818.875,A -85,B 0,C 180,E1 7425.944,E2 7425.944} C_VEL
LIN {X 0,Y 178.046,Z 808.623,A -85,B 0,C 180,E1 7419.706,E2 7419.706} C_VEL
LIN {X 0,Y 189.124,Z 797.967,A -85,B 0,C 180,E1 7414.972,E2 7414.972} C_VEL
LIN {X 0,Y 200.625,Z 786.318,A -85,B 0,C 180,E1 7410.999,E2 7410.999} C_VEL
LIN {X 0,Y 214.478,Z 770.979,A -85,B 0,C 180,E1 7407.079,E2 7407.079} C_VEL
LIN {X 0,Y 225.474,Z 757.607,A -85,B 0,C 180,E1 7404.466,E2 7404.466} C_VEL
LIN {X 0,Y 237.398,Z 741.689,A -85,B 0,C 180,E1 7402.015,E2 7402.015} C_VEL
LIN {X 0,Y 248.894,Z 724.201,A -85,B 0,C 180,E1 7399.949,E2 7399.949} C_VEL
LIN {X 0,Y 258.664,Z 707.456,A -85,B 0,C 180,E1 7398.387,E2 7398.387} C_VEL
LIN {X 0,Y 269.068,Z 686.847,A -85,B 0,C 180,E1 7396.894,E2 7396.894} C_VEL
LIN {X 0,Y 276.987,Z 668.176,A -85,B 0,C 180,E1 7395.851,E2 7395.851} C_VEL
LIN {X 0,Y 284.178,Z 648.094,A -85,B 0,C 180,E1 7394.984,E2 7394.984} C_VEL
LIN {X 0,Y 290.483,Z 625.4,A -85,B 0,C 180,E1 7394.274,E2 7394.274} C_VEL
LIN {X 0,Y 294.773,Z 604.604,A -85,B 0,C 180,E1 7393.775,E2 7393.775} C_VEL
LIN {X 0,Y 298.508,Z 574.894,A -85,B 0,C 180,E1 7393.199,E2 7393.199} C_VEL
LIN {X 0,Y 307.384,Z 489.628,A -85,B 0,C 180,E1 7391.635,E2 7391.635} C_VEL
LIN {X 0,Y 305.347,Z 485.259,A -85,B 0,C 180,E1 7389.043,E2 7389.043} C_VEL
LIN {X 0,Y 304.304,Z 482.998,A -85,B 0,C 180,E1 7387.362,E2 7387.362} C_VEL
LIN {X 0,Y 303.055,Z 480.015,A -85,B 0,C 180,E1 7384.542,E2 7384.542} C_VEL
LIN {X 0,Y 302.18,Z 478.631,A -85,B 0,C 180,E1 7379.81,E2 7379.81} C_VEL
LIN {X 0,Y 303.033,Z 479.996,A -85,B 0,C 180,E1 7375.079,E2 7375.079} C_VEL
LIN {X 0,Y 303.652,Z 481.602,A -85,B 0,C 180,E1 7373.477,E2 7373.477} C_VEL
LIN {X 0,Y 305.131,Z 484.693,A -85,B 0,C 180,E1 7370.855,E2 7370.855} C_VEL
LIN {X 0,Y 309.268,Z 491.765,A -85,B 0,C 180,E1 7366.158,E2 7366.158} C_VEL
LIN {X 0,Y 314.267,Z 496.964,A -85,B 0,C 180,E1 7362.407,E2 7362.407} C_VEL
LIN {X 0,Y 317.853,Z 499.643,A -85,B 0,C 180,E1 7360.235,E2 7360.235} C_VEL
LIN {X 0,Y 322.905,Z 503.873,A -85,B 0,C 180,E1 7357.036,E2 7357.036} C_VEL
LIN {X 0,Y 326.639,Z 506.347,A -85,B 0,C 180,E1 7354.43,E2 7354.43} C_VEL
LIN {X 0,Y 329.047,Z 507.896,A -85,B 0,C 180,E1 7352.59,E2 7352.59} C_VEL
LIN {X 0,Y 332.167,Z 511.149,A -85,B 0,C 180,E1 7349.822,E2 7349.822} C_VEL
LIN {X 0,Y 335.59,Z 514.009,A -85,B 0,C 180,E1 7346.347,E2 7346.347} C_VEL
LIN {X 0,Y 337.259,Z 515.252,A -85,B 0,C 180,E1 7344.613,E2 7344.613} C_VEL
LIN {X 0,Y 339.93,Z 518.521,A -85,B 0,C 180,E1 7341.638,E2 7341.638} C_VEL
LIN {X 0,Y 343.322,Z 521.265,A -85,B 0,C 180,E1 7337.946,E2 7337.946} C_VEL
LIN {X 0,Y 345.17,Z 522.531,A -85,B 0,C 180,E1 7335.852,E2 7335.852} C_VEL
LIN {X 0,Y 348.075,Z 526.106,A -85,B 0,C 180,E1 7332.174,E2 7332.174} C_VEL
LIN {X 0,Y 350.858,Z 528.362,A -85,B 0,C 180,E1 7328.663,E2 7328.663} C_VEL
LIN {X 0,Y 353.468,Z 529.997,A -85,B 0,C 180,E1 7325.165,E2 7325.165} C_VEL
LIN {X 0,Y 355.557,Z 532.886,A -85,B 0,C 180,E1 7321.87,E2 7321.87} C_VEL
LIN {X 0,Y 357.855,Z 535.022,A -85,B 0,C 180,E1 7318.176,E2 7318.176} C_VEL
LIN {X 0,Y 359.809,Z 536.26,A -85,B 0,C 180,E1 7314.634,E2 7314.634} C_VEL
LIN {X 0,Y 361.729,Z 537.101,A -85,B 0,C 180,E1 7310.889,E2 7310.889} C_VEL
LIN {X 0,Y 362.875,Z 538.828,A -85,B 0,C 180,E1 7307.809,E2 7307.809} C_VEL
LIN {X 0,Y 364.08,Z 540.464,A -85,B 0,C 180,E1 7304.309,E2 7304.309} C_VEL
LIN {X 0,Y 364.96,Z 541.533,A -85,B 0,C 180,E1 7300.736,E2 7300.736} C_VEL
LIN {X 0,Y 365.715,Z 542.145,A -85,B 0,C 180,E1 7297.225,E2 7297.225} C_VEL
LIN {X 0,Y 366.074,Z 542.507,A -85,B 0,C 180,E1 7293.602,E2 7293.602} C_VEL
LIN {X 0,Y 366.284,Z 542.626,A -85,B 0,C 180,E1 7290.156,E2 7290.156} C_VEL
LIN {X 0,Y 366.088,Z 542.508,A -85,B 0,C 180,E1 7286.555,E2 7286.555} C_VEL
LIN {X 0,Y 365.756,Z 542.188,A -85,B 0,C 180,E1 7283.092,E2 7283.092} C_VEL
LIN {X 0,Y 365.02,Z 541.602,A -85,B 0,C 180,E1 7279.535,E2 7279.535} C_VEL
LIN {X 0,Y 364.204,Z 540.622,A -85,B 0,C 180,E1 7276.182,E2 7276.182} C_VEL
LIN {X 0,Y 362.996,Z 539.013,A -85,B 0,C 180,E1 7272.529,E2 7272.529} C_VEL
LIN {X 0,Y 361.851,Z 537.233,A -85,B 0,C 180,E1 7269.457,E2 7269.457} C_VEL
LIN {X 0,Y 359.914,Z 536.312,A -85,B 0,C 180,E1 7265.549,E2 7265.549} C_VEL
LIN {X 0,Y 357.938,Z 535.082,A -85,B 0,C 180,E1 7261.97,E2 7261.97} C_VEL
LIN {X 0,Y 355.659,Z 532.999,A -85,B 0,C 180,E1 7258.285,E2 7258.285} C_VEL
LIN {X 0,Y 353.546,Z 530.126,A -85,B 0,C 180,E1 7254.964,E2 7254.964} C_VEL
LIN {X 0,Y 352.232,Z 529.169,A -85,B 0,C 180,E1 7253.177,E2 7253.177} C_VEL
LIN {X 0,Y 349.43,Z 527.324,A -85,B 0,C 180,E1 7249.495,E2 7249.495} C_VEL
LIN {X 0,Y 346.471,Z 524.346,A -85,B 0,C 180,E1 7245.835,E2 7245.835} C_VEL
LIN {X 0,Y 344.54,Z 521.966,A -85,B 0,C 180,E1 7243.454,E2 7243.454} C_VEL
LIN {X 0,Y 341.597,Z 520.007,A -85,B 0,C 180,E1 7240.188,E2 7240.188} C_VEL
LIN {X 0,Y 338.281,Z 516.628,A -85,B 0,C 180,E1 7236.493,E2 7236.493} C_VEL
LIN {X 0,Y 336.538,Z 514.562,A -85,B 0,C 180,E1 7234.573,E2 7234.573} C_VEL
LIN {X 0,Y 332.753,Z 511.693,A -85,B 0,C 180,E1 7230.756,E2 7230.756} C_VEL
LIN {X 0,Y 329.465,Z 508.38,A -85,B 0,C 180,E1 7227.765,E2 7227.765} C_VEL
LIN {X 0,Y 327.889,Z 506.987,A -85,B 0,C 180,E1 7226.437,E2 7226.437} C_VEL
LIN {X 0,Y 323.657,Z 504.44,A -85,B 0,C 180,E1 7223.485,E2 7223.485} C_VEL
LIN {X 0,Y 319.018,Z 500.695,A -85,B 0,C 180,E1 7220.454,E2 7220.454} C_VEL
LIN {X 0,Y 315.683,Z 497.937,A -85,B 0,C 180,E1 7218.465,E2 7218.465} C_VEL
LIN {X 0,Y 310.098,Z 492.914,A -85,B 0,C 180,E1 7214.566,E2 7214.566} C_VEL
LIN {X 0,Y 306.986,Z 488.269,A -85,B 0,C 180,E1 7211.555,E2 7211.555} C_VEL
LIN {X 0,Y 304.493,Z 483.318,A -85,B 0,C 180,E1 7208.117,E2 7208.117} C_VEL
LIN {X 0,Y 303.108,Z 480.062,A -85,B 0,C 180,E1 7205.11,E2 7205.11} C_VEL
LIN {X 0,Y 302.181,Z 478.635,A -85,B 0,C 180,E1 7200.379,E2 7200.379} C_VEL
LIN {X 0,Y 302.783,Z 479.741,A -85,B 0,C 180,E1 7196.213,E2 7196.213} C_VEL
LIN {X 0,Y 303.336,Z 480.651,A -85,B 0,C 180,E1 7194.704,E2 7194.704} C_VEL
